(* Check Setup Level with active key switch and an active movement *)
	IF xReset THEN
		xReset:=FALSE;
		xActivateOverlayMessage:=FALSE;
	END_IF;
	IF NOT(xActivateOverlayMessage) THEN
		xActiveSetupLevel:=	(T_Visu.ptrT_ExchgParam^.T_Visu.bActivSpecialLayer <> 0) AND
							T_StartUp.T_State.xCompleted AND NOT(T_StartUp.T_State.xBlockChangeMovementVisu);
		xDoNotCheckMovement:=	NOT(T_Process.xEnd) AND NOT(T_Process.xError) AND ((T_Process.iFunctNr = 10) OR (T_Process.iFunctNr = 20) OR (T_Process.iFunctNr = 30));
		xActiveProcess:=		NOT(T_Process.xEnd) AND NOT(T_Process.xError) AND (T_Process.iFunctNr = 40);
		xActiveStation:=		NOT(T_Station.TControl.xEnd) AND NOT(T_Station.TControl.xError) AND NOT(xActiveProcess) AND NOT(xDoNotCheckMovement);
		xActiveHWStation:=	T_Station.TControl.xActiveMovement AND NOT(xActiveProcess) AND NOT(xActiveStation) AND NOT(xDoNotCheckMovement);
		(* check if the ToolTorque was activatet *)
		xStopAxisWithStationFunction:=FALSE;
		IF xActiveHWStation THEN
			IF (T_Visu.T_PlcParam.dwActualPage = 220) THEN
				xActiveHWStation:=FALSE;
				xStopAxisWithStationFunction:=TRUE;
			END_IF;
		END_IF;
	END_IF;
	FallingEdgeKeySwitchOff(CLK:=xKeySwitch);
	IF xActiveSetupLevel THEN
		IF FallingEdgeKeySwitchOff.Q THEN
			IF xActiveProcess OR xActiveStation OR xActiveHWStation OR xStopAxisWithStationFunction THEN
				xActivateOverlayMessage:=TRUE;
				iStepSwitchMachineLevel:=1;
			END_IF;
		END_IF;
	END_IF;
(*
	IF NOT(xBlockChecking) THEN
		xActivateOverlayMessage:= xActivateOverlayMessage AND NOT
								(T_Station.TControl.xSecurityCircuitOff OR T_Station.TControl.xSecurityCircuitOn);
	END_IF;
*)
	IF xActivateOverlayMessage THEN
		CASE iStepSwitchMachineLevel OF
		1:	TONWaitTimeStateMachine(IN:=FALSE);
			(* next step *)
			iStepSwitchMachineLevel:=10;
		10:	TONWaitTimeStateMachine(IN:=TRUE,PT:=T#150ms);
			IF TONWaitTimeStateMachine.Q THEN
				TONWaitTimeStateMachine(IN:=FALSE);
				(* next step *)
				iStepSwitchMachineLevel:=20;
			END_IF;
		20:	IF T_TwinSafeOut.QxContactor_K3 AND T_TwinSafeOut.QxContactor_K4 THEN
				xPowerSupplyActive:=TRUE;
				T_Visu.ptrT_ExchgParam^.T_Visu.T_Message.iState:=121;	(* Display message -> The Movement of the machine will be breaked! *)
				(* with switching off of the key switch the power supply is not switched off and the movement are still active *)
				IF xActiveProcess THEN
					T_Process.xStop:=TRUE;
					iStepSwitchMachineLevel:=30;
				END_IF;
				IF xActiveStation THEN
					T_Station.TControl.xStop:=TRUE;
					iStepSwitchMachineLevel:=40;
				END_IF;
				IF xActiveHWStation THEN
					iStepSwitchMachineLevel:=60;
				END_IF;
				IF xStopAxisWithStationFunction THEN
					iStepSwitchMachineLevel:=70;
				END_IF;
			ELSE
				(* with switching off of the key switch the power supply is switched off *)
				xPowerSupplyActive:=FALSE;
				(* next step *)
				iStepSwitchMachineLevel:=80;
			END_IF;
		30:	IF T_Process.xEnd THEN
				(* next step *)
				iStepSwitchMachineLevel:=80;
			END_IF;
			IF NOT(T_TwinSafeOut.QxContactor_K3) OR NOT(T_TwinSafeOut.QxContactor_K4) THEN
				xPowerSupplyActive:=FALSE;
				iStepSwitchMachineLevel:=80;
			END_IF;
			T_Visu.ptrT_ExchgParam^.T_Visu.T_Message.iState:=121;	(* Display message -> The Movement of the machine will be breaked! *)
		40:	IF T_Station.TControl.xEnd THEN
				(* next step *)
				T_Station.TControl.xStop:=FALSE;
				iStepSwitchMachineLevel:=60;
			END_IF;
			IF NOT(T_TwinSafeOut.QxContactor_K3) OR NOT(T_TwinSafeOut.QxContactor_K4) THEN
				xPowerSupplyActive:=FALSE;
				iStepSwitchMachineLevel:=80;
			END_IF;
			T_Visu.ptrT_ExchgParam^.T_Visu.T_Message.iState:=121;	(* Display message -> The Movement of the machine will be breaked! *)
		60:	IF T_Station.THardware.TAxisToolLeft.T_CtrleSingle.xDone AND NOT(T_Station.THardware.TAxisToolLeft.T_CtrleSingle.xErr) THEN
				T_Station.THardware.TAxisToolLeft.T_CtrleSingle.iFunction:=5;
				T_Station.THardware.TAxisToolLeft.T_CtrleSingle.xExecute:=TRUE;
			END_IF;
			IF NOT(T_Station.THardware.TAxisToolLeft.T_CtrleSingle.xDone) AND T_Station.THardware.TAxisToolLeft.T_CtrleSingle.xNotMoving AND NOT(T_Station.THardware.TAxisToolLeft.T_CtrleSingle.xErr) THEN
				T_Station.THardware.TAxisToolLeft.T_CtrleSingle.xReset:=TRUE;
			END_IF;
			IF T_Station.THardware.TAxisToolRight.T_CtrleSingle.xDone AND NOT(T_Station.THardware.TAxisToolRight.T_CtrleSingle.xErr) THEN
				T_Station.THardware.TAxisToolRight.T_CtrleSingle.iFunction:=5;
				T_Station.THardware.TAxisToolRight.T_CtrleSingle.xExecute:=TRUE;
			END_IF;
			IF NOT(T_Station.THardware.TAxisToolRight.T_CtrleSingle.xDone) AND T_Station.THardware.TAxisToolRight.T_CtrleSingle.xNotMoving AND NOT(T_Station.THardware.TAxisToolRight.T_CtrleSingle.xErr) THEN
				T_Station.THardware.TAxisToolRight.T_CtrleSingle.xReset:=TRUE;
			END_IF;
			IF T_Station.THardware.TAxisToolCenter.T_CtrleSingle.xDone AND NOT(T_Station.THardware.TAxisToolCenter.T_CtrleSingle.xErr) THEN
				T_Station.THardware.TAxisToolCenter.T_CtrleSingle.iFunction:=5;
				T_Station.THardware.TAxisToolCenter.T_CtrleSingle.xExecute:=TRUE;
			END_IF;
			IF NOT(T_Station.THardware.TAxisToolCenter.T_CtrleSingle.xDone) AND T_Station.THardware.TAxisToolCenter.T_CtrleSingle.xNotMoving AND NOT(T_Station.THardware.TAxisToolCenter.T_CtrleSingle.xErr) THEN
				T_Station.THardware.TAxisToolCenter.T_CtrleSingle.xReset:=TRUE;
			END_IF;
			IF T_Station.THardware.TAxisToolFeeder.T_CtrleSingle.xDone AND NOT(T_Station.THardware.TAxisToolFeeder.T_CtrleSingle.xErr) THEN
				T_Station.THardware.TAxisToolFeeder.T_CtrleSingle.iFunction:=5;
				T_Station.THardware.TAxisToolFeeder.T_CtrleSingle.xExecute:=TRUE;
			END_IF;
			IF NOT(T_Station.THardware.TAxisToolFeeder.T_CtrleSingle.xDone) AND NOT(T_Station.THardware.TAxisToolFeeder.T_CtrleSingle.xNotMoving) AND NOT(T_Station.THardware.TAxisToolFeeder.T_CtrleSingle.xErr) THEN
				T_Station.THardware.TAxisToolFeeder.T_CtrleSingle.iFunction:=5;
				T_Station.THardware.TAxisToolFeeder.T_CtrleSingle.xExecute:=TRUE;
			END_IF;
			IF NOT(T_Station.THardware.TAxisToolFeeder.T_CtrleSingle.xDone) AND T_Station.THardware.TAxisToolFeeder.T_CtrleSingle.xNotMoving AND NOT(T_Station.THardware.TAxisToolFeeder.T_CtrleSingle.xErr) THEN
				T_Station.THardware.TAxisToolFeeder.T_CtrleSingle.xReset:=TRUE;
			END_IF;
			IF T_Station.THardware.TAxisGrindFeeder.T_CtrleSingle.xDone AND NOT(T_Station.THardware.TAxisGrindFeeder.T_CtrleSingle.xErr) THEN
				T_Station.THardware.TAxisGrindFeeder.T_CtrleSingle.iFunction:=5;
				T_Station.THardware.TAxisGrindFeeder.T_CtrleSingle.xExecute:=TRUE;
			END_IF;
			IF NOT(T_Station.THardware.TAxisGrindFeeder.T_CtrleSingle.xDone) AND NOT(T_Station.THardware.TAxisGrindFeeder.T_CtrleSingle.xNotMoving) AND NOT(T_Station.THardware.TAxisGrindFeeder.T_CtrleSingle.xErr) THEN
				T_Station.THardware.TAxisGrindFeeder.T_CtrleSingle.iFunction:=5;
				T_Station.THardware.TAxisGrindFeeder.T_CtrleSingle.xExecute:=TRUE;
			END_IF;
			IF NOT(T_Station.THardware.TAxisGrindFeeder.T_CtrleSingle.xDone) AND T_Station.THardware.TAxisGrindFeeder.T_CtrleSingle.xNotMoving AND NOT(T_Station.THardware.TAxisGrindFeeder.T_CtrleSingle.xErr) THEN
				T_Station.THardware.TAxisGrindFeeder.T_CtrleSingle.xReset:=TRUE;
			END_IF;
			IF NOT(T_Station.THardware.TCylToolTension.T_CtrleCyl.xDone) THEN T_Station.THardware.TCylToolTension.T_CtrleCyl.xReset:=TRUE; END_IF;
			T_Visu.ptrT_ExchgParam^.T_Visu.T_Message.iState:=121;	(* Display message -> The Movement of the machine will be breaked! *)
			(* next step *)
			iStepSwitchMachineLevel:=80;
		70:	IF T_Station.TControl.xEnd THEN
				(* next step *)
				T_Station.TControl.iFunctNr:=3;
				T_Station.TControl.xStart:=TRUE;
				iStepSwitchMachineLevel:=71;
			END_IF;
			IF NOT(T_TwinSafeOut.QxContactor_K3) OR NOT(T_TwinSafeOut.QxContactor_K4) THEN
				xPowerSupplyActive:=FALSE;
				iStepSwitchMachineLevel:=80;
			END_IF;
			T_Visu.ptrT_ExchgParam^.T_Visu.T_Message.iState:=121;	(* Display message -> The Movement of the machine will be breaked! *)
		71:	IF NOT(T_Station.TControl.xStart) AND T_Station.TControl.xEnd THEN
				(* next step *)
				iStepSwitchMachineLevel:=80;
			END_IF;
			IF NOT(T_TwinSafeOut.QxContactor_K3) OR NOT(T_TwinSafeOut.QxContactor_K4) THEN
				xPowerSupplyActive:=FALSE;
				iStepSwitchMachineLevel:=80;
			END_IF;
		80:	IF NOT(T_Visu.T_CtrleVisu.xExecute) AND T_Visu.T_CtrleVisu.xDone THEN
				T_Visu.ptrT_ExchgParam^.T_Visu.T_Message.iState:=0;
				T_Visu.ptrT_ExchgParam^.T_Visu.bActivSpecialLayer:=0;
				T_Visu.ptrT_ExchgParam^.T_TouchScreenBtPanel.iStateBtLeft:=0;
				T_Visu.ptrT_ExchgParam^.T_TouchScreenNavPanel.wState:=1;
				T_Visu.T_PlcParam.dwSetNewPage:=16#A;	(* Main Page wird aufgerufen *)
				T_Visu.T_CtrleVisu.iFunction:=1;
				T_Visu.T_CtrleVisu.xExecute:=TRUE;
				iStepSwitchMachineLevel:=90;
			END_IF;
		90:	IF NOT(T_Visu.T_CtrleVisu.xExecute) AND T_Visu.T_CtrleVisu.xDone THEN
				T_StartUp.T_State.xBlockChangeMovementVisu:=TRUE;	(* Lock the navigation of the visu *)
				T_Visu.ptrT_ExchgParam^.T_SafetyCtrl.xBlockVisuObject:=TRUE;
				T_StartUp.T_State.xBlockVisuNavigation:=FALSE;	(* Unlock the navigation of the visu *)
				T_Visu.ptrT_ExchgParam^.T_SafetyCtrl.bStateAutoGeometry:=1;
				T_Visu.ptrT_ExchgParam^.T_SafetyCtrl.bStateAutoGroove:=1;
				T_Visu.ptrT_ExchgParam^.T_SafetyCtrl.bStateReference:=1;
				T_Visu.ptrT_ExchgParam^.T_SafetyCtrl.bStateToolCalibration:=1;
				T_Visu.ptrT_ExchgParam^.T_SafetyCtrl.bStateToolTorque:=1;
				T_Visu.ptrT_ExchgParam^.T_SafetyCtrl.bStateTeachInToolLeft:=1;
				T_Visu.ptrT_ExchgParam^.T_SafetyCtrl.bStateTeachInToolCenter:=1;
				T_Visu.ptrT_ExchgParam^.T_SafetyCtrl.bStateTeachInToolRight:=1;
				T_Visu.ptrT_ExchgParam^.T_SafetyCtrl.bStateTeachInToolFeeder:=1;
				T_Visu.ptrT_ExchgParam^.T_SafetyCtrl.bStateTeachInGrindFeeder:=1;
				T_Visu.ptrT_ExchgParam^.T_StationCommon.iWireFeederRefIndexState:=1;
				(* Overlay Message Error *)
				T_Visu.ptrT_ExchgParam^.T_SafetyCtrl.bStateMessageError:=1;
				T_Visu.ptrT_ExchgParam^.T_SafetyCtrl.bStateMessageInfo:=0;
				T_Visu.ptrT_ExchgParam^.T_SafetyCtrl.bStateMessageWarning:=0;
				IF xPowerSupplyActive THEN
					T_Visu.ptrT_ExchgParam^.T_SafetyCtrl.iMsgErrorLine1:=18;	(* WHILE A MOVEMENT THE KEY SWITCH *)
					T_Visu.ptrT_ExchgParam^.T_SafetyCtrl.iMsgErrorLine2:=18;	(* HAS BEEN SWITCHED OFF! *)
					T_Visu.ptrT_ExchgParam^.T_SafetyCtrl.iMsgErrorLine3:=18;	(* NOW YOU ARE ON THE NORMAL OPERATION *)
					T_Visu.ptrT_ExchgParam^.T_SafetyCtrl.iMsgErrorLine4:=18;	(* AND THE POWER SUPPLY IS STILL SWITCHED ON *)
					T_Visu.ptrT_ExchgParam^.T_SafetyCtrl.xConfirmMsgError:=FALSE;
				ELSE
					T_Visu.ptrT_ExchgParam^.T_SafetyCtrl.iMsgErrorLine1:=17;	(* WHILE A MOVEMENT THE KEY SWITCH *)
					T_Visu.ptrT_ExchgParam^.T_SafetyCtrl.iMsgErrorLine2:=17;	(* HAS BEEN SWITCHED OFF! *)
					T_Visu.ptrT_ExchgParam^.T_SafetyCtrl.iMsgErrorLine3:=17;	(* NOW YOU ARE ON THE NORMAL OPERATION *)
					T_Visu.ptrT_ExchgParam^.T_SafetyCtrl.iMsgErrorLine4:=17;	(* AND THE POWER SUPPLY IS SWITCHED OFF *)
					T_Visu.ptrT_ExchgParam^.T_SafetyCtrl.xConfirmMsgError:=FALSE;
				END_IF;
				(* next step *)
				iStepSwitchMachineLevel:=100;
			END_IF;
		100:	IF T_Visu.ptrT_ExchgParam^.T_SafetyCtrl.xConfirmMsgError THEN
				T_StartUp.T_State.xBlockChangeMovementVisu:=FALSE;	(* Unlock the navigation of the visu *)
				T_Visu.ptrT_ExchgParam^.T_SafetyCtrl.xBlockVisuObject:=FALSE;
				T_StartUp.T_State.xBlockVisuNavigation:=FALSE;	(* Unlock the navigation of the visu *)
				T_Visu.ptrT_ExchgParam^.T_SafetyCtrl.bStateAutoGeometry:=1;
				T_Visu.ptrT_ExchgParam^.T_SafetyCtrl.bStateAutoGroove:=1;
				T_Visu.ptrT_ExchgParam^.T_SafetyCtrl.bStateReference:=1;
				T_Visu.ptrT_ExchgParam^.T_SafetyCtrl.bStateToolCalibration:=1;
				T_Visu.ptrT_ExchgParam^.T_SafetyCtrl.bStateToolTorque:=1;
				T_Visu.ptrT_ExchgParam^.T_SafetyCtrl.bStateTeachInToolLeft:=1;
				T_Visu.ptrT_ExchgParam^.T_SafetyCtrl.bStateTeachInToolCenter:=1;
				T_Visu.ptrT_ExchgParam^.T_SafetyCtrl.bStateTeachInToolRight:=1;
				T_Visu.ptrT_ExchgParam^.T_SafetyCtrl.bStateTeachInToolFeeder:=1;
				T_Visu.ptrT_ExchgParam^.T_SafetyCtrl.bStateTeachInGrindFeeder:=1;
				T_Visu.ptrT_ExchgParam^.T_StationCommon.iWireFeederRefIndexState:=1;
				T_Visu.ptrT_ExchgParam^.T_SafetyCtrl.bStateMessageError:=0;
				T_Visu.ptrT_ExchgParam^.T_SafetyCtrl.xConfirmMsgError:=FALSE;
				xActivateOverlayMessage:=FALSE;
				iStepSwitchMachineLevel:=1;
			END_IF;
			IF NOT(T_TwinSafeOut.QxContactor_K3) OR NOT(T_TwinSafeOut.QxContactor_K4) THEN
				T_Visu.ptrT_ExchgParam^.T_SafetyCtrl.iMsgErrorLine1:=17;	(* WHILE A MOVEMENT THE KEY SWITCH *)
				T_Visu.ptrT_ExchgParam^.T_SafetyCtrl.iMsgErrorLine2:=17;	(* HAS BEEN SWITCHED OFF! *)
				T_Visu.ptrT_ExchgParam^.T_SafetyCtrl.iMsgErrorLine3:=17;	(* NOW YOU ARE ON THE NORMAL OPERATION *)
				T_Visu.ptrT_ExchgParam^.T_SafetyCtrl.iMsgErrorLine4:=17;	(* AND THE POWER SUPPLY IS SWITCHED OFF *)
			END_IF;
			IF T_TwinSafeOut.QxContactor_K3 AND T_TwinSafeOut.QxContactor_K4  THEN
				T_Visu.ptrT_ExchgParam^.T_SafetyCtrl.iMsgErrorLine1:=18;	(* WHILE A MOVEMENT THE KEY SWITCH *)
				T_Visu.ptrT_ExchgParam^.T_SafetyCtrl.iMsgErrorLine2:=18;	(* HAS BEEN SWITCHED OFF! *)
				T_Visu.ptrT_ExchgParam^.T_SafetyCtrl.iMsgErrorLine3:=18;	(* NOW YOU ARE ON THE NORMAL OPERATION *)
				T_Visu.ptrT_ExchgParam^.T_SafetyCtrl.iMsgErrorLine4:=18;	(* AND THE POWER SUPPLY IS STILL SWITCHED ON *)
			END_IF;
		END_CASE;
	END_IF;
END_FUNCTION_BLOCK

(* POU PRG_VISU_LAYER5/PRG_VISU, FBD *)
PROGRAM PRG_VISU
VAR
	fbVisuQVis: FBQVIS;
	xSecurityKey: BOOL;
	FBCtrleButton: FB_CTRLEBUTTON;
END_VAR
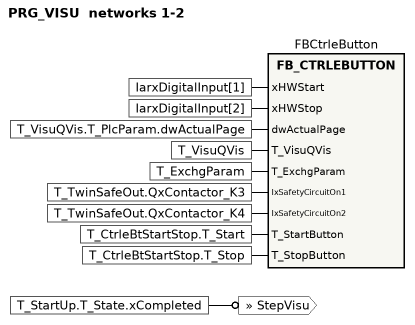
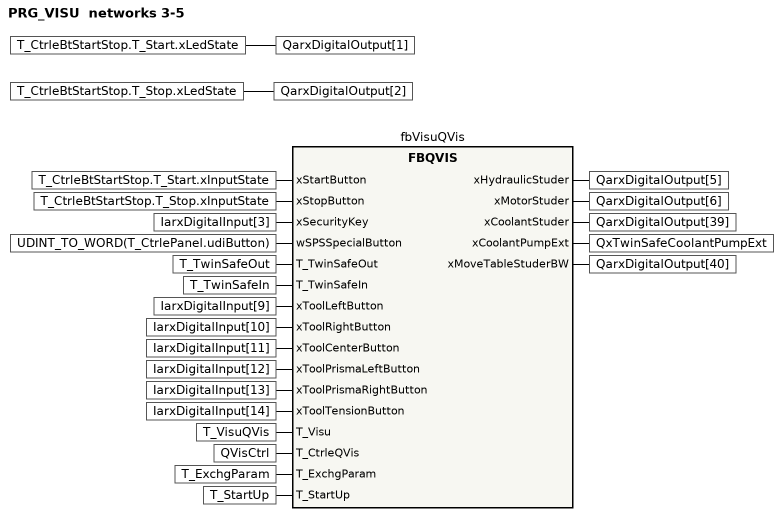
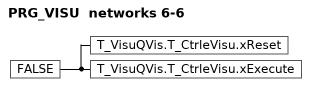
_FBD_ (* Function Block Diagram *)
NETWORK 1 (* VISUALISATION LEVEL-->LAYER 5 *)
	FBCtrleButton:FB_CTRLEBUTTON(xHWStart: IarxDigitalInput[1], xHWStop: IarxDigitalInput[2], dwActualPage: T_VisuQVis.T_PlcParam.dwActualPage, T_VisuQVis: T_VisuQVis, T_ExchgParam: T_ExchgParam, IxSafetyCircuitOn1: T_TwinSafeOut.QxContactor_K3, IxSafetyCircuitOn2: T_TwinSafeOut.QxContactor_K4, T_StartButton: T_CtrleBtStartStop.T_Start, T_StopButton: T_CtrleBtStartStop.T_Stop)
NETWORK 2
	NOT T_StartUp.T_State.xCompleted => >>StepVisu
NETWORK 3
	T_CtrleBtStartStop.T_Start.xLedState => QarxDigitalOutput[1]
NETWORK 4
	T_CtrleBtStartStop.T_Stop.xLedState => QarxDigitalOutput[2]
NETWORK 5 StepVisu:
	fbVisuQVis:FBQVIS(xStartButton: T_CtrleBtStartStop.T_Start.xInputState, xStopButton: T_CtrleBtStartStop.T_Stop.xInputState, xSecurityKey: IarxDigitalInput[3], wSPSSpecialButton: UDINT_TO_WORD(T_CtrlePanel.udiButton), T_TwinSafeOut: T_TwinSafeOut, T_TwinSafeIn: T_TwinSafeIn, xToolLeftButton: IarxDigitalInput[9], xToolRightButton: IarxDigitalInput[10], xToolCenterButton: IarxDigitalInput[11], xToolPrismaLeftButton: IarxDigitalInput[12], xToolPrismaRightButton: IarxDigitalInput[13], xToolTensionButton: IarxDigitalInput[14], T_Visu: T_VisuQVis, T_CtrleQVis: QVisCtrl, T_ExchgParam: T_ExchgParam, T_StartUp: T_StartUp, xMotorStuder => QarxDigitalOutput[6], xCoolantStuder => QarxDigitalOutput[39], xCoolantPumpExt => QxTwinSafeCoolantPumpExt, xMoveTableStuderBW => QarxDigitalOutput[40]) => QarxDigitalOutput[5]
NETWORK 6
	FALSE => T_VisuQVis.T_CtrleVisu.xReset, T_VisuQVis.T_CtrleVisu.xExecute
_END_FBD_
(* the same logic as Structured Text *)
(* Network 1: VISUALISATION LEVEL-->LAYER 5 *)
FBCtrleButton(xHWStart := IarxDigitalInput[1], xHWStop := IarxDigitalInput[2], dwActualPage := T_VisuQVis.T_PlcParam.dwActualPage, T_VisuQVis := T_VisuQVis, T_ExchgParam := T_ExchgParam, IxSafetyCircuitOn1 := T_TwinSafeOut.QxContactor_K3, IxSafetyCircuitOn2 := T_TwinSafeOut.QxContactor_K4, T_StartButton := T_CtrleBtStartStop.T_Start, T_StopButton := T_CtrleBtStartStop.T_Stop);
(* Network 2 *)
IF NOT T_StartUp.T_State.xCompleted THEN JMP StepVisu; END_IF;
(* Network 3 *)
QarxDigitalOutput[1] := T_CtrleBtStartStop.T_Start.xLedState;
(* Network 4 *)
QarxDigitalOutput[2] := T_CtrleBtStartStop.T_Stop.xLedState;
(* Network 5 *)
StepVisu:
fbVisuQVis(xStartButton := T_CtrleBtStartStop.T_Start.xInputState, xStopButton := T_CtrleBtStartStop.T_Stop.xInputState, xSecurityKey := IarxDigitalInput[3], wSPSSpecialButton := UDINT_TO_WORD(T_CtrlePanel.udiButton), T_TwinSafeOut := T_TwinSafeOut, T_TwinSafeIn := T_TwinSafeIn, xToolLeftButton := IarxDigitalInput[9], xToolRightButton := IarxDigitalInput[10], xToolCenterButton := IarxDigitalInput[11], xToolPrismaLeftButton := IarxDigitalInput[12], xToolPrismaRightButton := IarxDigitalInput[13], xToolTensionButton := IarxDigitalInput[14], T_Visu := T_VisuQVis, T_CtrleQVis := QVisCtrl, T_ExchgParam := T_ExchgParam, T_StartUp := T_StartUp);
QarxDigitalOutput[6] := fbVisuQVis.xMotorStuder;
QarxDigitalOutput[39] := fbVisuQVis.xCoolantStuder;
QxTwinSafeCoolantPumpExt := fbVisuQVis.xCoolantPumpExt;
QarxDigitalOutput[40] := fbVisuQVis.xMoveTableStuderBW;
QarxDigitalOutput[5] := fbVisuQVis.xHydraulicStuder;
(* Network 6 *)
T_VisuQVis.T_CtrleVisu.xReset := FALSE;
T_VisuQVis.T_CtrleVisu.xExecute := FALSE;
END_PROGRAM

(* POU PRG_VISU_LAYER5/FB_VISU/FBQVIS, ST *)
FUNCTION_BLOCK FBQVIS
VAR_INPUT
	xStartButton:BOOL;					(* external start button *)
	xStopButton:BOOL;					(* external stop button *)
	xSecurityKey:BOOL;					(* state of the keyswitch *)
	wSPSSpecialButton:WORD;			(* input of the special button of the controlpanel *)
	T_TwinSafeOut:ST_TWINSAFE_OUT;	(* Output of the TwinSAFE components *)
	T_TwinSafeIn:ST_TWINSAFE_IN;		(* Input of the TwinSAFE components *)
(*22.12.2009: KFS	{	*)
	xToolLeftButton:BOOL;					(* Signal of the button for closing the ToolLeft-->this is only for the MicroRod *)
	xToolRightButton:BOOL;				(* Signal of the button for closing the ToolRight-->this is only for the MicroRod *)
	xToolCenterButton:BOOL;				(* Signal of the button for closing the ToolCenter-->this is only for the MicroRod *)
	xToolPrismaLeftButton:BOOL;			(* Signal of the button for closing the ToolPrismaLeft-->this is only for the MicroRod *)
	xToolPrismaRightButton:BOOL;			(* Signal of the button for closing the ToolPrismaRight-->this is only for the MicroRod *)
	xToolTensionButton:BOOL;				(* Signal of the button for activate the ToolTension-->this is only for the MicroRod *)
(*22.12.2009: KFS	}	*)
END_VAR
VAR_OUTPUT
(* SOA 02.02.2023     {     *)
	xHydraulicStuder: 	BOOL;  					(*Hydraulic Pump of Studer S20 Machine*)
	xMotorStuder: BOOL;						(*Grinding-Engine of Studer S20 Machine*)
	xCoolantStuder: BOOL;						(*Coolant Pump of Studer S20 Machine*)
	xCoolantPumpExt: BOOL;					(*Coolant Pump external*)
	xMoveTableStuderBW:BOOL;
(* SOA 02.02.2023    }   *)
END_VAR
VAR_IN_OUT
	T_Visu:ST_QVIS;
	T_CtrleQVis:ST_QVISCTRLE;
	T_ExchgParam:ST_QVIS_EXCHG_PARAM;
	T_StartUp:ST_STARTUP;
END_VAR
VAR
	RisingEdgeActiv:R_TRIG;
	RisingEdgeExecute:R_TRIG;
	RisingEdgeExecuteAction:R_TRIG;
	RisingEdgeBtPanelLeft:R_TRIG;
	FallingEdgeBtPanelLeft:F_TRIG;
	RisingEdgeSpecialLayer:R_TRIG;
	FallingEdgeSpecialLayer:F_TRIG;
	RisingEdgeTouchScreenNavPanel:R_TRIG;
	FallingEdgeTouchScreenNavPanel:F_TRIG;
	RisingEdgeBtPanelRight:R_TRIG;
	FallingEdgeBtPanelRight:F_TRIG;
	RisingEdgeBtFunctionPanel:R_TRIG;
	FallingEdgeBtFunctionPanel:F_TRIG;
	RisingEdgeDynPassword:R_TRIG;
	RisingEdgeGeometryManagement:R_TRIG;
	RisingEdgeToolDiameter:R_TRIG;
	RisingEdgePrisma:R_TRIG;
	xChangePage:BOOL:=FALSE;
	dwInCount_QVisCmd:DWORD:=0;
	xTmp: BOOL;
	wActivBtLeft: WORD;
	wActivBtRight: WORD;
	fbQvisInitPage:FBQVIS_INITPAGE;
	xNavPanelChangePage: BOOL;
	xBtPanelLeftChangePage:BOOL;
	xBtPanelRightChangePage: BOOL; (*SOA*)
	xNextPageVertical:BOOL;
	xSetParameterPage:BOOL;
	xActivationSection1: BOOL;
	xActivationSection2: BOOL;
	xActivationSection3: BOOL;
	xActivationSection4: BOOL;
	xActivationSection5: BOOL; (*SOA *)
	xActivationSection6: BOOL; (*SOA *)

	xSetPitchEqual: BOOL;
	iStepAction: INT;
	xStepActionDone: BOOL;
	bOldActivSpecialLayer: BYTE;
	wSpecialLayerGeneralActivTask: WORD;
	wSpecialLayerToolRotActivTask: WORD;
	wSpecialLayerWireFeedActivTask: WORD;
	wSpecialLayerGrindAxisActivTask: WORD;
	wSpecialLayerGeneralActivPage: WORD;
	wSpecialLayerToolRotActivPage: WORD;
	wSpecialLayerWireFeedActivPage: WORD;
	wSpecialLayerGrindAxisActivPage: WORD;
	dwSetNewPage: DWORD;
	wNormalLayerActivTask: WORD;
	wNormalLayerActivPage: WORD;
	ii: INT;
	wTmp: WORD;
	awNormalLayerActivPage:ARRAY [1..6] OF WORD;
	awSpecialLayerGeneralActivPage:ARRAY [1..6] OF WORD;
	awSpecialLayerToolRotActivPage:ARRAY [1..6] OF WORD;
	awSpecialLayerWireFeedActivPage:ARRAY [1..6] OF WORD;
	awSpecialLayerGrindAxisActivPage:ARRAY [1..6] OF WORD;
	wTmpNormalLayerActivTask: WORD;
	wTmpSpecialLayerGeneralActivTask: WORD;
	wTmpSpecialLayerToolRotActivTask: WORD;
	wTmpSpecialLayerWireFeedActivTask: WORD;
	wTmpSpecialLayerGrindAxisActivTask: WORD;
	wStandardPageNr: WORD;
	iTmpActivBtLeft: INT;
	(* Random *)
	fbGetCpuAccount:GETCPUCOUNTER;
	fbPwSystem:FBPW_SYSTEM;
	(* Pw *)
	iPwSystem:INT;
	iStepCounter: INT;
	arSaveToolGeometry:ST_GEOMETRY;
	rSectionPitch: REAL;
	ptxActiveSection1: POINTER TO BOOL;
	ptxActiveSection2: POINTER TO BOOL;
	ptxActiveSection3: POINTER TO BOOL;
	ptxActiveSection4: POINTER TO BOOL;
	ptxActiveSection5: POINTER TO BOOL;
	ptxActiveSection6: POINTER TO BOOL;

	xOverlayMeasureToolDia: BOOL;
	xPlungeActivation: BOOL;
	xDisplaceActivation: BOOL;
	xCorrectionToolDiameterAdd: BOOL;
	xCorrectionToolDiameterAddMore: BOOL;
	xCorrectionToolDiameterSub: BOOL;
	xCorrectionToolDiameterSubMore: BOOL;
	xResetToolDiameterCorrection: BOOL;
	xKeyPadActivation: BOOL;
	xFctCorrectionToolDiameter: BOOL;
	rCorrectionValue: REAL;

(* Key panel button "Esc"/"Enter" *)
	RisingEdgeKeyPanel_Esc:R_TRIG;
	RisingEdgeKeyPanel_Enter:R_TRIG;
(*22.12.2009: KFS	{	 *)
(* External button for the tool-clamping*)
	RisingEdgeBtToolLeft:R_TRIG;
	RisingEdgeBtToolRight:R_TRIG;
	RisingEdgeBtToolCenter:R_TRIG;
	RisingEdgeBtToolPrismaLeft:R_TRIG;
	RisingEdgeBtToolPrismaRight:R_TRIG;
	RisingEdgeBtToolTension:R_TRIG;
(*22.12.2009: KFS	}	 *)
(* variable start action *)
	TimerAction:TON;
	TimerNotReady:TOF;
	tTimeOutAction:TIME;
	xSelectPrisma: BOOL;
	xToolTensForceAdd: BOOL;
	xToolTensForceAddMore: BOOL;
	xToolTensForceSub: BOOL;
	xToolTensForceSubMore: BOOL;
	xResetCalculToolRotTorque: BOOL;
	rCalcTotalToolLength: REAL;
	xTmpSecurityKey: BOOL;
	RisingEdgeTemp:R_TRIG;
	TONWAIT: TON;
	xPart1: BOOL;
	xPart2: BOOL;
	xPart3: BOOL;
	xPart4: BOOL;
	xPart5: BOOL;
	xPart6: BOOL;

	iPartActive: INT;
	xToolRotationMasterSlave: BOOL;
	xSwitchMasterSlave: BOOL;
	xQvisActiv: BOOL;
	TimerQVis: TON;
	RisingEdgeReset:R_TRIG;
	xConfirmResetFB: BOOL;
	xFirstRead: BOOL;
	ptrTeachINAxis:POINTER TO ST_AXIS;
	ptrCylAction:POINTER TO ST_CYLINDER;
	xStopAxis: BOOL;
	xMoveRelPosition: BOOL;
	TParaAxisTeachIN:ST_EXCHG_PARAM_TEACHIN;
	xMoveContinousVel: BOOL;
	xMoveAbsPosition: BOOL;
	bButtonPanelLocked: BYTE;
	xDelayActionBtPanelRight: BOOL;
	TimerPressBtPanelRight: TON;

(* Structure page *)
	T_ConfigPage:ST_CONFIGPAGE;
	wMaskBtPanelLeft: WORD;
	wMaskBtPanelRight: WORD;
	wMaskFunctionPanel: WORD;
	RisingEdgeProcessDone: R_TRIG;
	xStopImmediatly: BOOL;
	RisingEdgeProcessError: R_TRIG;
	RisingEdgeResetProcess: R_TRIG;
	RisingEdgeExecuteProcess: R_TRIG;
	RisingEdgeActionNotReady: R_TRIG;
	FallingEdgeActionNotReady: F_TRIG;
	RisingEdgeActionDone: R_TRIG;
	xBlockConfirmMessage: BOOL;
	RisingEdgeActionError: R_TRIG;
	RisingEdgeResetAction: R_TRIG;
	xSlowFast: BOOL;
	iSelectedAxis: INT;
	xSlowFastJogToolRotation: BOOL;
	xSlowFastJogToolFeeder: BOOL;
	xSlowFastJogGrindFeeder: BOOL;
	xToggleAxisPower: BOOL;
	xResetAxis: BOOL;
	xUpdateProfileList: BOOL;
	jj: INT;
	RisingEdgePtrProfileListUpDown: R_TRIG;
	iPointerListProfile: INT;
	iActualActiveProfile: INT;
	xAction_CopyProfileToProcess: BOOL;
	xProfileFileNotFound: BOOL;
	iToLoadProfileNr: INT;
	sToLoadProfileName: STRING;
	sTmpDynamicText: STRING;
	xAction_LoadProfileToProcessImage: BOOL;
	xAction_SaveNovRAM: BOOL;
	xActionDeleteProfile: BOOL;
	TimerONTmp: TON;
	iStepActionNovRam: INT;
	xAction_SaveProfileToFile: BOOL;
	iTmp: INT;
	sTmp: STRING;
	sTmp_2: STRING;
	RisingEdgeTimeOut: R_TRIG;
	fbCompareProfileProcessValue:FB_COMPAREPROFILEPROCESSVALUE;
	FailingEdgeGeometryManagement: F_TRIG;
	FailingEdgePrisma: F_TRIG;
	rCalcMinMaxToolDia: REAL;
	xResetParaListValue: BOOL;
	xActivateStationFunction: BOOL;
	iTmpStationFunctionNr: INT;
	xFirstReadInit: BOOL;
	xFirstReadReset: BOOL;
	xMicroRodActive: BOOL;
	FBCalcTorqueToolLeft: FB_CALC_TORQUE;
	FBCalcTorqueToolCenter: FB_CALC_TORQUE;
	FBCalcTorqueToolRight: FB_CALC_TORQUE;
	xTmpStopAxis: BOOL;
	RisingEdgeStartButton: R_TRIG;
	dwPageNrProcessStart: DWORD;
	FallingEdgeStartButton: F_TRIG;
	RisingEdgeStopButton: R_TRIG;
	FallingEdgeStopButton: F_TRIG;
	xToggleCylinderState: BOOL;
	dwTmpActualPage: DWORD;
	xUpdateErrorList: BOOL;
	RisingEdgeErrorList: R_TRIG;
	xParameterSavedErrorList: BOOL;
	xDeleteErrorList: BOOL;
	FBQVisErrorList: FBQVIS_ERROR_LIST;
	FBSetErrorList:FB_SETERRORLIST;
	xProcessMachine: BOOL;
	xProcessStation: BOOL;
	iStepProcess: INT;
	xStepProcessDone: BOOL;
	xStopProcess: BOOL;
	xAction_StopCycle: BOOL;
	xWaitStopEnd: BOOL;
	xWaitStopCycleEnd: BOOL;
	iStepWaitStopEnd: INT;
	xActionProcStation: BOOL;
	xActionProcMachine: BOOL;
	RisingEdgeKeySwitch1: R_TRIG;
	FailingEdgeKeySwitch1: F_TRIG;
	TimerDisplayMessage: TON;
	RisingEdgeReleaseWarning: R_TRIG;
	rCalcPrismaFactor: REAL;
	xFirstReadParaList: BOOL;
	iTmpSelectParaList: INT;
	xAction_SaveNovRAMWithoutConfirm: BOOL;
	diErrorNr: DINT;
	FBErrorMessage : FB_ErrorMessage;
	fbQvisClearError:FBQVIS_CLEARERROR;
	xResetError: BOOL;
	TONTimeWaitMsg: TON;
	xCheckQuitError: BOOL;
	bStateMachine: BYTE;
	xSetStateMachine: BOOL;
	iSelectAxisToolRotation: INT;
	rAutoTimeTotal: REAL;
	rToolRotationSpeed: REAL;
	iAutoProcess: INT;
	xBlockGrindFeederActivation: BOOL;
	xToolFeederMoveStartPos: BOOL;
	xToggleAllAxisPower: BOOL;
	FBCalcProcessTime: FB_CALCPROCESSTIME;
	xReferenceAxis: BOOL;
	xTeachPosition: BOOL;
	xCalcAngleRefIndex: BOOL;
	uiToolLeftZeroTorque: UINT;
	uiToolCenterZeroTorque: UINT;
	uiToolRightZeroTorque: UINT;
	xSetCalculToolRotTorque: BOOL;
	rActualToolFeederPosition: REAL;
	xReadActualToolFeedPos: BOOL;
	xReadActualToolFeedPos1: BOOL;
	rActualToolFeederPosition1: REAL;
	rToolTotalLength: REAL;
	xCalcFirstTime: BOOL;
	xFirstReadParaList1: BOOL;
	iTmpSelectParaList1: INT;
	xTmpTeach: BOOL;
	wTmpActivBtRight: WORD;
	xOverlayGrindFeedSetPlung: BOOL;
	xOpenMessageBox: BOOL;
	lrActualGrindFeedPosition: LREAL;
	lrToWriteGrindFeedPosition: LREAL;
	xCalcAgainProcTime: BOOL;
	xToolFeederMoveLoadPos: BOOL;
	xWarmUp:BOOL;
	iSelectedCylinder: INT;
	xWarmUpMessage: BOOL;
	xWarmUpMessageActiv: BOOL;
	xWarmUpMessageDone: BOOL;

(*SOA 12.01.2023 { *)
	(*WarmUp*)
	xSaveValueWarmUp: BOOL;
	fbSetLocalTime	:NT_SetLocalTime;
	fbGetSysTime	: NT_GetTime;
	xGetTime: BOOL;
        TIMESTR :TIMESTRUCT;
	TONWaitGetTime: TON;
	xSaveTimeAndDate: BOOL;
	xInitReadFirstTimeTimeStamp: BOOL;
	iCountDayOfWeek: INT;
	xReadyToCheckWarmUp: BOOL;
	wCheckTimeWarmUp: WORD;
	wConvertMinute: WORD;
	wConertMinute_StartTime: WORD;
	wCheckTimeWarmUp_StartTime: WORD;
	wConertMinute_StopTime: WORD;
	wCheckTimeWarmUp_StopTime: WORD;
	xReadyToStartNextTime: BOOL;
	xWarmuUp_Start: BOOL;
	xWarmUp_Stop: BOOL;
	TONWarmUpChangeColour: TON;

	TONDelayMessage: TON;
	xConfirmStartWarmUp: BOOL;
	xStartUpConfirmed: BOOL;
	xStopWarmup: BOOL;
(*SOA 12.01.2023 { *)


	(* .CtrlFunctionButton *)
	wForceMaskFunctionPanel:WORD;						(* IGS *)
	aiForceRTrigActionFunctionPanel:ARRAY [1..12] OF INT;	(* IGS *)
	aiDelectRTrigActionFunctionPanel:ARRAY [1..12] OF INT;	(* IGS *)

	(* .CtrlVisuFunction *)
	xCWCCW:BOOL;										(* IGS *)
	xCylBrake:BOOL;										(* IGS *)
END_VAR
(****************************************************************************************************************************************************)
(******    This Functionblock manages the hole visualisation. It is the interface from QVis and the control application         	  *******)
(****************************************************************************************************************************************************)
	IF NOT(xFirstRead) THEN
		xFirstRead:=TRUE;
		T_Visu.ptrT_ExchgParam:=ADR(T_ExchgParam);
	END_IF;
	RisingEdgeActiv(CLK:=T_Visu.T_CtrleVisu.xActive);
	IF RisingEdgeActiv.Q THEN
		(* call functionblock init. *)
		fbQvisInitPage(T_Visu:=T_Visu);
		(* Init. variable for visualisation action *)
		T_Visu.T_CtrleAction.xDone:=TRUE;
		T_Visu.T_CtrleAction.xExecute:=FALSE;
		T_Visu.T_CtrleAction.xNotReady:=FALSE;
		T_Visu.T_CtrleAction.xErr:=FALSE;
		T_Visu.T_CtrleAction.udiErrorID:=0;
		T_Visu.T_CtrleVisu.xDone:=FALSE;
		T_Visu.ptrT_ExchgParam:=ADR(T_ExchgParam);
		wNormalLayerActivTask:=1;
		wSpecialLayerGeneralActivTask:=1;
		wSpecialLayerToolRotActivTask:=1;
		wSpecialLayerWireFeedActivTask:=1;
		wSpecialLayerGrindAxisActivTask:=1;
		wNormalLayerActivPage:=10;
		wSpecialLayerGeneralActivPage:=110;
		wSpecialLayerToolRotActivPage:=210;
		wSpecialLayerWireFeedActivPage:=310;
		wSpecialLayerGrindAxisActivPage:=410;
		T_Visu.ptrT_ExchgParam^.T_TouchScreenNavPanel.wState:=1;
		wStandardPageNr:=10;
		T_Visu.ptrT_ExchgParam^.T_Visu.T_Level.iPwSystem:=999;
		wTmpNormalLayerActivTask:=1;
		wTmpSpecialLayerGeneralActivTask:=1;
		wTmpSpecialLayerToolRotActivTask:=1;
		wTmpSpecialLayerWireFeedActivTask:=1;
		wTmpSpecialLayerGrindAxisActivTask:=1;
		FOR ii:=1 TO 6 DO
			awNormalLayerActivPage[ii]:=wStandardPageNr;
			wStandardPageNr:=wStandardPageNr + 10;
		END_FOR;
		wStandardPageNr:=110;
		FOR ii:=1 TO 6 DO
			awSpecialLayerGeneralActivPage[ii]:=wStandardPageNr;
			wStandardPageNr:=wStandardPageNr + 10;
		END_FOR;
		wStandardPageNr:=210;
		FOR ii:=1 TO 6 DO
			awSpecialLayerToolRotActivPage[ii]:=wStandardPageNr;
			wStandardPageNr:=wStandardPageNr + 10;
		END_FOR;
		wStandardPageNr:=310;
		FOR ii:=1 TO 6 DO
			awSpecialLayerWireFeedActivPage[ii]:=wStandardPageNr;
			wStandardPageNr:=wStandardPageNr + 10;
		END_FOR;
		wStandardPageNr:=410;
		FOR ii:=1 TO 6 DO
			awSpecialLayerGrindAxisActivPage[ii]:=wStandardPageNr;
			wStandardPageNr:=wStandardPageNr + 10;
		END_FOR;
		IF NOT(xFirstReadInit) THEN
			xFirstReadInit:=TRUE;
			T_Visu.T_PlcParam.dwSetNewPage:=1001;
		ELSE
			T_Visu.T_PlcParam.dwSetNewPage:=0;
		END_IF;
		T_Visu.T_PlcParam.dwActualPage:=0;
		T_Visu.T_PlcParam.dwPreviousPage:=0;
		iPointerListProfile:=1;
		iActualActiveProfile:=-1;
		TimerAction(IN:=FALSE);
		(* Init FB *)
		fbQvisClearError(	xExecute:=FALSE,
						iError:=0,
						T_Message:=T_ExchgParam.T_Visu.T_Message,
						T_Station:=T_Station,
						T_Process:=T_Process,
						T_NovRAM:=T_NovRAM,
						T_Profile:=T_Profile,
						T_HDD:=T_HDD,
						xDone=>T_Visu.T_CtrleAction.xDone,
						xNotReady=>T_Visu.T_CtrleAction.xNotReady,
						xErr=>T_Visu.T_CtrleAction.xErr,
						udiErrorID=>T_Visu.T_CtrleAction.udiErrorID);
		T_Visu.ptrT_ExchgParam^.T_Cylinder.iSelectToolTensionForce:=1;	(* For starting the machine always set  the process force for the ToolTension *)
		ptrTeachINAxis:=ADR(T_Station.THardware.TAxisToolLeft);
	END_IF;

	IF NOT (T_Visu.T_CtrleVisu.xActive) THEN
		RETURN;
	END_IF;

(* waiting for reset *)
	RisingEdgeReset(CLK:=T_Visu.T_CtrleVisu.xReset);
	IF RisingEdgeReset.Q THEN
		(* Init. structure *)
		T_Visu.T_CtrleVisu.xDone:=FALSE;
		T_Visu.T_CtrleVisu.iFunction:=0;
		T_Visu.T_CtrleVisu.xErr:=FALSE;
		T_Visu.T_CtrleVisu.udiErrorID:=0;
		IF NOT(xFirstReadReset) THEN
			xFirstReadReset:=TRUE;
			T_Visu.T_PlcParam.dwSetNewPage:=1001;
		ELSE
			T_Visu.T_PlcParam.dwSetNewPage:=0;
		END_IF;
		T_Visu.T_PlcParam.dwActualPage:=0;
		T_Visu.T_PlcParam.dwPreviousPage:=0;
		T_Visu.ptrT_ExchgParam^.T_Visu.iQVisActivNewPage:=0;
		wNormalLayerActivTask:=1;
		wSpecialLayerGeneralActivTask:=1;
		wSpecialLayerToolRotActivTask:=1;
		wSpecialLayerWireFeedActivTask:=1;
		wSpecialLayerGrindAxisActivTask:=1;
		wNormalLayerActivPage:=10;
		wSpecialLayerGeneralActivPage:=110;
		wSpecialLayerToolRotActivPage:=210;
		wSpecialLayerWireFeedActivPage:=310;
		wSpecialLayerGrindAxisActivPage:=410;
		wTmpNormalLayerActivTask:=1;
		wTmpSpecialLayerGeneralActivTask:=1;
		wTmpSpecialLayerToolRotActivTask:=1;
		wTmpSpecialLayerWireFeedActivTask:=1;
		wTmpSpecialLayerGrindAxisActivTask:=1;
		T_Visu.ptrT_ExchgParam^.T_TouchScreenNavPanel.wState:=1;
		T_Visu.ptrT_ExchgParam^.T_Visu.bActivSpecialLayer:=0;
		T_Visu.ptrT_ExchgParam^.T_TouchScreenBtPanel.iStateBtLeft:=0;
		wStandardPageNr:=10;
		T_Visu.ptrT_ExchgParam^.T_Visu.T_Level.iPwSystem:=999;
		FOR ii:=1 TO 6 DO
			awNormalLayerActivPage[ii]:=wStandardPageNr;
			wStandardPageNr:=wStandardPageNr + 10;
		END_FOR;
		wStandardPageNr:=110;
		FOR ii:=1 TO 6 DO
			awSpecialLayerGeneralActivPage[ii]:=wStandardPageNr;
			wStandardPageNr:=wStandardPageNr + 10;
		END_FOR;
		wStandardPageNr:=210;
		FOR ii:=1 TO 6 DO
			awSpecialLayerToolRotActivPage[ii]:=wStandardPageNr;
			wStandardPageNr:=wStandardPageNr + 10;
		END_FOR;
		wStandardPageNr:=310;
		FOR ii:=1 TO 6 DO
			awSpecialLayerWireFeedActivPage[ii]:=wStandardPageNr;
			wStandardPageNr:=wStandardPageNr + 10;
		END_FOR;
		wStandardPageNr:=410;
		FOR ii:=1 TO 6 DO
			awSpecialLayerGrindAxisActivPage[ii]:=wStandardPageNr;
			wStandardPageNr:=wStandardPageNr + 10;
		END_FOR;
		(* Activ reset structure control action *)
		T_Visu.T_CtrleAction.xReset:=TRUE;
		(* Activ reset structure control process *)
		T_Visu.T_CtrleProcess.xReset:=TRUE;
		(* Init. pw value *)
		T_Visu.ptrT_ExchgParam^.T_Visu.T_Level.iPwSystem:=999;
		(* Init. Error *)
		T_Visu.ptrT_ExchgParam^.T_Visu.T_Message.iState:=0;
		T_Visu.ptrT_ExchgParam^.T_Visu.T_Message.sDynamicTextEnglish:='';
		T_Visu.ptrT_ExchgParam^.T_Visu.T_Message.sDynamicTextDeutsch:='';
		T_Visu.ptrT_ExchgParam^.T_Visu.T_Message.sDynamicTextFrancais:='';
		T_Visu.ptrT_ExchgParam^.T_TouchScreenBtPanel.iStateBtLeft:=0;
		T_Visu.ptrT_ExchgParam^.T_Cylinder.iSelectCylinder_Sonder1:=1;
		T_Visu.ptrT_ExchgParam^.T_StationCommon.iWireFeederAngleRefIndex:=0;
		T_Visu.ptrT_ExchgParam^.T_TeachIn.iSelectAxisGrind:=1;
		T_Visu.ptrT_ExchgParam^.T_TeachIn.iSelectAxisToolRotation:=1;
		T_Visu.ptrT_ExchgParam^.T_TeachIn.iSelectAxisWireFeeder:=1;
		T_Visu.ptrT_ExchgParam^.T_TeachIn.xSlowFastToolRotation:=FALSE;
		T_Visu.ptrT_ExchgParam^.T_TeachIn.xSlowFastToolFeed:=FALSE;
		T_Visu.ptrT_ExchgParam^.T_TeachIn.xSlowFastGrindFeeder:=FALSE;
		T_Visu.ptrT_ExchgParam^.T_InfoValueCommon.rToolTensionForce:=T_NovRAM.T_Data.T_ProcessImageData.T_ProcessPara.rToolTensionProcess;
		(* active confirmation *)
		xConfirmResetFB:=TRUE;
		(* exit function bloc *)
		RETURN;
	ELSE
		IF xConfirmResetFB THEN
			(* confirm reset FB *)
			T_Visu.T_CtrleVisu.xDone:=TRUE;
			T_Visu.T_CtrleVisu.xErr:=FALSE;
			T_Visu.T_CtrleVisu.udiErrorID:=0;
			(* reset variable *)
			xConfirmResetFB:=FALSE;
			(* activ research if Qvis is activ *)
			xQvisActiv:=TRUE;
			T_Visu.T_CtrleVisu.xQvis:=FALSE;
			dwInCount_QVisCmd:=T_CtrleQVis.dwInCount;
		END_IF
	END_IF

(* determin if qvis activ *)
	IF xQvisActiv THEN
		(* timer time off  *)
		TimerQVis(IN:=TRUE,PT:=T#2s);
		IF dwInCount_QVisCmd = T_CtrleQVis.dwInCount THEN
			(* Init. command *)
			T_CtrleQVis.dwInCommand:=1;
			T_CtrleQVis.dwInQVisCtrlAddress:=ADR(T_CtrleQVis);
			T_CtrleQVis.dwInParameterAddress:=ADR(T_Visu.T_PlcParam.dwSetNewPage);
			(* start command *)
			T_CtrleQVis.dwInCount:=T_CtrleQVis.dwInCount+1;
			(* Activ Timer *)
			TimerQVis(IN:=FALSE);
		ELSE
			IF T_CtrleQVis.dwInCount = T_CtrleQVis.dwOutCount THEN
			(* command done *)
				IF T_CtrleQVis.diOutStatus = 0 THEN
				(* command done without error *)
					xQvisActiv:=FALSE;
					T_Visu.T_CtrleVisu.xQvis:=TRUE;
					T_Visu.T_PlcParam.dwActualPage:=T_Visu.T_PlcParam.dwSetNewPage;
				END_IF
			ELSE
			(* test time off, restart command *)
				IF TimerQVis.Q THEN
					dwInCount_QVisCmd:=T_CtrleQVis.dwInCount;
				END_IF
			END_IF
		END_IF
	END_IF

(* exit FB if Qvis inactiv *)
	IF NOT(T_Visu.T_CtrleVisu.xQvis) THEN RETURN; END_IF

	IF (T_Visu.T_PlcParam.dwActualPage > 0) AND (T_Visu.T_PlcParam.dwActualPage <= 999) THEN
		(* copy config page structure *)
		T_ConfigPage:=T_Visu.T_ConfigPage[T_Visu.T_PageIndex[T_Visu.T_PlcParam.dwActualPage].iIndexConfigPage];
		T_Visu.ptrT_ExchgParam^. T_TouchScreenNavPanel.wNotMasktext:=T_ConfigPage.wMaskTouchScreenNavPanel;
		T_Visu.ptrT_ExchgParam^.T_TouchScreenBtPanel.iNotMaskTextBt:=16#0;
		T_Visu.ptrT_ExchgParam^.T_TouchScreenBtPanel.iNotMaskTextBt:=WORD_TO_INT(INT_TO_WORD(T_Visu.ptrT_ExchgParam^.T_TouchScreenBtPanel.iNotMaskTextBt) OR T_ConfigPage.wMaskBtPanelRight);
		T_Visu.ptrT_ExchgParam^.T_TouchScreenBtPanel.iNotMaskTextBt:=WORD_TO_INT(INT_TO_WORD(T_Visu.ptrT_ExchgParam^.T_TouchScreenBtPanel.iNotMaskTextBt) OR T_ConfigPage.wMaskBtPanelLeft);
		T_Visu.ptrT_ExchgParam^.T_TouchScreenBtPanel.iNotMaskTextBt:=WORD_TO_INT(NOT(INT_TO_WORD(T_Visu.ptrT_ExchgParam^.T_TouchScreenBtPanel.iNotMaskTextBt)));
	END_IF;

(* monitor page Errorlist for Machine *)
	xTmp:=	(T_Visu.T_PlcParam.dwActualPage = 60) OR
			(T_Visu.T_PlcParam.dwActualPage = 160) OR
			(T_Visu.T_PlcParam.dwActualPage = 260) OR
			(T_Visu.T_PlcParam.dwActualPage = 360) OR
			(T_Visu.T_PlcParam.dwActualPage = 460);
	IF xTmp THEN
		(* Check if Station will be changed without changing the Error Page *)
		IF (dwTmpActualPage <> T_Visu.T_PlcParam.dwActualPage) THEN
			xUpdateErrorList:=TRUE;
			dwTmpActualPage:=T_Visu.T_PlcParam.dwActualPage;
		END_IF;
	END_IF;
	IF xTmp OR xUpdateErrorList THEN
		IF NOT(xTmp) AND xUpdateErrorList THEN
			RisingEdgeErrorList(CLK:=xUpdateErrorList);
		ELSE
			RisingEdgeErrorList(CLK:=xTmp AND NOT(xUpdateErrorList));
		END_IF;
		xUpdateErrorList:=FALSE;
		IF RisingEdgeErrorList.Q THEN
			FBQVisErrorList(	T_ErrorList:= T_ErrorList,
							T_ErrorNrList:= T_NovRAM.T_Data.T_ErrorNrList,
							T_MsgErrorEnglish:= T_Visu.ptrT_ExchgParam^.T_Visu.T_MsgErrorEnglish,
							T_MsgErrorDeutsch:= T_Visu.ptrT_ExchgParam^.T_Visu.T_MsgErrorDeutsch,
							T_MsgErrorFrancais:= T_Visu.ptrT_ExchgParam^.T_Visu.T_MsgErrorFrancais);
		END_IF;
	ELSE
		RisingEdgeErrorList(CLK:=FALSE);
	END_IF;

(* Refresh Errorlist for Machine and Station *)
	FBSetErrorList(	TControlStation:= T_Station.TControl,
					TProcess:= T_Process,
					xParameterSaved:= xParameterSavedErrorList,
					T_ErrorNrList:= T_NovRAM.T_Data.T_ErrorNrList,
					xSetForceError:= T_Visu.ptrT_ExchgParam^.T_SafetyCtrl.xSetForceError,
					diSetForceErrorNr:= T_Visu.ptrT_ExchgParam^.T_SafetyCtrl.diSetForceErrorNr);
	IF FBSetErrorList.xSaveParameter THEN
		IF T_Visu.T_CtrleAction.xDone AND NOT(T_Visu.T_CtrleAction.xExecute) AND T_NovRAM.T_Ctrle.xDone AND NOT(T_NovRAM.T_Ctrle.xExecute) THEN
			xParameterSavedErrorList:=TRUE;
			xUpdateErrorList:=TRUE;
			T_NovRAM.T_Ctrle.xExecute:=TRUE;
			T_NovRAM.T_Ctrle.iFunction:=2;
			T_NovRAM.T_Data.T_ErrorNrList;
		END_IF;
	END_IF;

(* Monitoring Visu Parameter *)
	T_Visu.ptrT_ExchgParam^.T_StationCommon.rConvertMaxToolLength:=T_NovRAM.T_Data.T_Standard.T_MachineConfig.rConfigMaxToolLength * 10.0;	(* convert from cm to mm *)
	T_Visu.ptrT_ExchgParam^.T_StationCommon.T_ParamToolTensionSystem.rMaxForceTT:=T_NovRAM.T_Data.T_Standard.T_ToolTensionSystem.rMaxForceTT;
	IF (T_NovRam.T_Data.T_Standard.T_MachineConfig.iConfigMachineType = 2) THEN
		xMicroRodActive:=TRUE;
	ELSE
		xMicroRodActive:=FALSE;
	END_IF;
	IF (T_Visu.T_PlcParam.dwActualPage = 170) AND ((T_Visu.ptrT_ExchgParam^.T_Config.iEditParam >= 120) AND (T_Visu.ptrT_ExchgParam^.T_Config.iEditParam <= 129)) THEN
		IF NOT(xFirstReadParaList) THEN
			iTmpSelectParaList:=T_Visu.ptrT_ExchgParam^.T_Config.iSelectParaList;
		END_IF;
		xFirstReadParaList:=TRUE;
		T_Visu.ptrT_ExchgParam^.T_Config.xBlockParaListNavi:=FALSE;
		T_Visu.ptrT_ExchgParam^.T_Config.xBlockParaListNavi1:=TRUE;
		T_Visu.ptrT_ExchgParam^.T_Config.xBlockProfilList:=FALSE;
		T_Visu.ptrT_ExchgParam^.T_Config.xBlockNavParaList:=FALSE;
		T_Visu.ptrT_ExchgParam^.T_Config.iEditParam:=iFctGetEditParaList(	dwActualPage:=120,
																	xMicroRodActive:=xMicroRodActive,
																	iSelectParaList:=T_Visu.ptrT_ExchgParam^.T_Config.iSelectParaList,
																	iSelectParaListTeachRot:=T_Visu.ptrT_ExchgParam^.T_Config.iSelectParaListTeachRot);
		(* 09.12.2010 KFS:	{	*)
		IF (T_ExchgParam.T_Visu.T_Level.iActLevel <>2) THEN
			IF  (T_Visu.ptrT_ExchgParam^.T_Config.iEditParam = 121) THEN
				 T_Visu.ptrT_ExchgParam^.T_Config.iEditParam:= 126;
			ELSIF ( T_Visu.ptrT_ExchgParam^.T_Config.iEditParam = 123) THEN
				 T_Visu.ptrT_ExchgParam^.T_Config.iEditParam:= 127;
			ELSIF ( T_Visu.ptrT_ExchgParam^.T_Config.iEditParam = 125) THEN
				 T_Visu.ptrT_ExchgParam^.T_Config.iEditParam:= 128;
			END_IF;
		END_IF;
		(* 09.12.2010 KFS:	}	*)
		IF (iTmpSelectParaList <> T_Visu.ptrT_ExchgParam^.T_Config.iSelectParaList) THEN
			iTmpSelectParaList:=T_Visu.ptrT_ExchgParam^.T_Config.iSelectParaList;
			xResetParaListValue:=TRUE;
		END_IF;
	ELSE
		xFirstReadParaList:=FALSE;
		T_Visu.ptrT_ExchgParam^.T_Config.xBlockNavParaList:=TRUE;
	END_IF;
	IF (T_Visu.T_PlcParam.dwActualPage = 270) AND ((T_Visu.ptrT_ExchgParam^.T_Config.iEditParam >= 210) AND (T_Visu.ptrT_ExchgParam^.T_Config.iEditParam <= 219)) THEN
		IF NOT(xFirstReadParaList1) THEN
			iTmpSelectParaList1:=T_Visu.ptrT_ExchgParam^.T_Config.iSelectParaListTeachRot;
		END_IF;
		xFirstReadParaList1:=TRUE;
		T_Visu.ptrT_ExchgParam^.T_Config.xBlockNavParaListTeachRot:=FALSE;
		T_Visu.ptrT_ExchgParam^.T_Config.iEditParam:=iFctGetEditParaList(	dwActualPage:=210,
																	xMicroRodActive:=xMicroRodActive,
																	iSelectParaList:=T_Visu.ptrT_ExchgParam^.T_Config.iSelectParaListTeachRot,
																	iSelectParaListTeachRot:=T_Visu.ptrT_ExchgParam^.T_Config.iSelectParaListTeachRot);
		IF (iTmpSelectParaList1 <> T_Visu.ptrT_ExchgParam^.T_Config.iSelectParaListTeachRot) THEN
			iTmpSelectParaList1:=T_Visu.ptrT_ExchgParam^.T_Config.iSelectParaListTeachRot;
			xResetParaListValue:=TRUE;
		END_IF;
	ELSE
		xFirstReadParaList1:=FALSE;
		T_Visu.ptrT_ExchgParam^.T_Config.xBlockNavParaListTeachRot:=TRUE;
	END_IF;
	xTmp:=	(T_Visu.T_PlcParam.dwActualPage = 170) OR
			(T_Visu.T_PlcParam.dwActualPage = 270) OR
			(T_Visu.T_PlcParam.dwActualPage = 370) OR
			(T_Visu.T_PlcParam.dwActualPage = 470);
	IF xTmp AND (T_Visu.ptrT_ExchgParam^.T_Config.iEditParam = 0) THEN
		T_Visu.ptrT_ExchgParam^.T_Config.xBlockParaListNavi:=TRUE;
		T_Visu.ptrT_ExchgParam^.T_Config.xBlockParaListNavi1:=TRUE;
	END_IF;

(* Monitor dynamic mask for button panel left and right and function panel *)
	IF T_Visu.T_CtrleProcess.xDone OR T_Visu.T_CtrleProcess.xErr THEN
	(* Set the standard mask *)
		wMaskBtPanelLeft:=T_ConfigPage.wMaskBtPanelLeft;
		wMaskBtPanelRight:=T_ConfigPage.wMaskBtPanelRight;
		wMaskFunctionPanel:=T_ConfigPage.wMaskFunctionPanel;
	(* Set the dynamic mask *)
	ELSE	wMaskBtPanelLeft:=T_ConfigPage.wMaskBtPanelLeft AND T_ConfigPage.wMaskActiveMachineBtPanelLeft;
			wMaskBtPanelRight:=T_ConfigPage.wMaskActiveMachineBtPanelRight;
			wMaskFunctionPanel:=T_ConfigPage.wMaskActiveMachineFunctionPanel;
	END_IF
	(* Check activ Page *)
	IF (T_Visu.T_PlcParam.dwActualPage = 170) OR (T_Visu.T_PlcParam.dwActualPage = 270) OR (T_Visu.T_PlcParam.dwActualPage = 370) OR (T_Visu.T_PlcParam.dwActualPage = 470) THEN
		IF (T_Visu.ptrT_ExchgParam^.T_Config.iEditParam = 0) THEN
			wMaskBtPanelRight:=16#0;
		END_IF;
		IF (T_Visu.ptrT_ExchgParam^.T_Config.iEditParam = 130) OR (T_Visu.ptrT_ExchgParam^.T_Config.iEditParam = 131) THEN
			wMaskBtPanelRight:=16#0;
		END_IF;
	END_IF;
	(* Config. divers mask *)
	T_Visu.ptrT_ExchgParam^.T_TouchScreenBtPanel.iNotMaskTextBt
	 :=(16#1F XOR wMaskBtPanelLeft) OR (16#3E0 XOR wMaskBtPanelRight);
	(* management Fn button panel availability *)
	T_Visu.ptrT_ExchgParam^.T_BtFunctionPanel.wNotMasktext:=16#FFF XOR wMaskFunctionPanel;
	(* management navigation panel mask *)
	T_Visu.ptrT_ExchgParam^.T_TouchScreenNavPanel.wNotMasktext:=T_ConfigPage.wMaskTouchScreenNavPanel;


MaskFunctionButton;

(************************************************************************************************************************************************************************)
(********start of the managment of the external start-stop button, special button and function button and task button and external tool buttons********)
(************************************************************************************************************************************************************************)
CtrlStartStopButton;
CtrlPanelLeftButton;
CtrlPanelRightButton;
CtrlFunctionButton;
CtrlTaskBar;
(************************************************************************************************************************************************************************)
(*********end of the managment of the external start-stop button, special button and function button and task button and external tool buttons********)
(************************************************************************************************************************************************************************)



(* set system level *)
	IF (T_Visu.ptrT_ExchgParam^.T_Visu.T_Level.iPwSystem <> 999) AND (T_Visu.T_PlcParam.dwActualPage = 40) THEN
		IF T_Visu.ptrT_ExchgParam^.T_Visu.T_Level.iPwSystem = iPwSystem THEN
		(* pw correct *)
			T_Visu.ptrT_ExchgParam^.T_Visu.T_Level.iActLevel:=2;
			T_Visu.ptrT_ExchgParam^.T_Visu.T_Message.iState:=2;
		(* wrong pw *)
		ELSE 	T_Visu.ptrT_ExchgParam^.T_Visu.T_Message.iState:=3; END_IF
		T_Visu.ptrT_ExchgParam^.T_Visu.T_Level.iPwSystem:=999;
	END_IF
	IF (T_Visu.T_PlcParam.dwActualPage = 40) THEN
		RisingEdgeDynPassword(CLK:=TRUE);
		IF RisingEdgeDynPassword.Q THEN
			fbGetCpuAccount;
			fbPwSystem(	dwCounter:=fbGetCpuAccount.fbGetCpuCounter.dwCpuCntHi+fbGetCpuAccount.fbGetCpuCounter.dwCpuCntLo,
						iRandom=>T_Visu.ptrT_ExchgParam^.T_Visu.T_Level.iRandom,
						iPwSystem=>iPwSystem);
		END_IF;
	ELSE
		RisingEdgeDynPassword(CLK:=FALSE);
	END_IF;

(************************************************************************************************************************************************************************)
(**********************************						Profile Management Start						****************************************)
(************************************************************************************************************************************************************************)

(* Update profile list *)
	IF xUpdateProfileList THEN
		xTmp:= 	iPointerListProfile > 0
				AND (iPointerListProfile+4) <= csiMaxProfile;
		IF xTmp THEN
			jj:=1;
			FOR ii:=iPointerListProfile TO iPointerListProfile+4 DO
				T_Visu.ptrT_ExchgParam^.T_ProfileCommon.T_ProfileList[jj].iNumber:=ii;
				T_Visu.ptrT_ExchgParam^.T_ProfileCommon.T_ProfileList[jj].sName:=T_NovRam.T_Data.T_IDProfileStation[ii].sName;
				jj:=jj+1;
			END_FOR
		END_IF
		(* confirm update *)
		xUpdateProfileList:=FALSE;
	END_IF

(* Compare Profile and Process value *)
	xTmp:=	(T_Visu.ptrT_ExchgParam^.T_StationCommon.T_InfoProcess.iProfile <> 0);
	IF xTmp THEN
		fbCompareProfileProcessValue(T_Data_ProcessImageLoadData:=T_NovRam.T_Data.T_ProcessImageLoadData,
									T_Data_ProcessImageData:=T_NovRam.T_Data.T_ProcessImageData,
									xMicroRodActive:=xMicroRodActive);
		T_Visu.ptrT_ExchgParam^.T_StationCommon.T_InfoProcess.xOnlineValueModified:=fbCompareProfileProcessValue.xProcessValueModified;
	END_IF

(* monitor change actual profile common *)
	IF (T_Visu.T_PlcParam.dwActualPage = 130) THEN
		IF T_Visu.ptrT_ExchgParam^.T_ProfileCommon.T_Id.iNumber<>iActualActiveProfile THEN
			IF T_Visu.T_CtrleAction.xDone THEN
				(* set value from selected profile *)
				T_Visu.ptrT_ExchgParam^.T_ProfileCommon.T_Id.sName
					:=T_NovRam.T_Data.T_IDProfileStation[T_Visu.ptrT_ExchgParam^.T_ProfileCommon.T_Id.iNumber].sName;
				(* save value from selected profile *)
				iActualActiveProfile:=T_Visu.ptrT_ExchgParam^.T_ProfileCommon.T_Id.iNumber;
			END_IF
		END_IF
	END_IF

(* Pointer Profile List Up/Down Slow *)
	RisingEdgePtrProfileListUpDown(CLK:=	T_Visu.ptrT_ExchgParam^.T_ProfileCommon.T_ProfileManage.xListProfileUp
										OR T_Visu.ptrT_ExchgParam^.T_ProfileCommon.T_ProfileManage.xListProfileDown);
	IF RisingEdgePtrProfileListUpDown.Q THEN
		IF T_Visu.ptrT_ExchgParam^.T_ProfileCommon.T_ProfileManage.xListProfileUp THEN
			iPointerListProfile:=iPointerListProfile-5;
		ELSE iPointerListProfile:=iPointerListProfile+5; END_IF
		(* min/max=1/6 *)
		IF iPointerListProfile>(csiMaxProfile -5) THEN iPointerListProfile:=(csiMaxProfile - 4); END_IF
		IF iPointerListProfile<0 THEN iPointerListProfile:=1; END_IF
		T_Visu.ptrT_ExchgParam^.T_ProfileCommon.T_ProfileManage.xListProfileUp:=FALSE;
		T_Visu.ptrT_ExchgParam^.T_ProfileCommon.T_ProfileManage.xListProfileDown:=FALSE;
		(* Update display  list *)
		xUpdateProfileList:=TRUE;
	END_IF

(* Pointer Profile List Up/Down Fast *)
	RisingEdgePtrProfileListUpDown(CLK:=	T_Visu.ptrT_ExchgParam^.T_ProfileCommon.T_ProfileManage.xListProfileUpFast
										OR T_Visu.ptrT_ExchgParam^.T_ProfileCommon.T_ProfileManage.xListProfileDownFast);
	IF RisingEdgePtrProfileListUpDown.Q THEN
		IF T_Visu.ptrT_ExchgParam^.T_ProfileCommon.T_ProfileManage.xListProfileUpFast THEN
			iPointerListProfile:=iPointerListProfile-10;
		ELSE iPointerListProfile:=iPointerListProfile+10; END_IF
		(* min/max=1/6 *)
		IF iPointerListProfile>(csiMaxProfile -5) THEN iPointerListProfile:=(csiMaxProfile - 4); END_IF
		IF iPointerListProfile<0 THEN iPointerListProfile:=1; END_IF
		T_Visu.ptrT_ExchgParam^.T_ProfileCommon.T_ProfileManage.xListProfileUpFast:=FALSE;
		T_Visu.ptrT_ExchgParam^.T_ProfileCommon.T_ProfileManage.xListProfileDownFast:=FALSE;
		(* Update display  list *)
		xUpdateProfileList:=TRUE;
	END_IF

(************************************************************************************************************************************************************************)
(**********************************						Profile Management End						****************************************)
(************************************************************************************************************************************************************************)

(* Display info or warning message *)
	RisingEdgeKeySwitch1(CLK:=xSecurityKey);
	FailingEdgeKeySwitch1(CLK:=xSecurityKey);
	IF T_Visu.ptrT_ExchgParam^.T_Visu.T_Message.iState <> 0 THEN
		(* info message *)
		IF T_Visu.ptrT_ExchgParam^.T_Visu.T_Message.iState < 100THEN
		(* activ message during 3s, after that the message will be cleared *)
			TimerDisplayMessage(IN:=TRUE,PT:=T#3s);
			IF TimerDisplayMessage.Q THEN
				T_Visu.ptrT_ExchgParam^.T_Visu.T_Message.iState:=0;
					T_ExchgParam.T_FunctionCommon.xWarmUp_MessageWarning_2:=FALSE;   (* SOA 20.02.2023 *)
				TimerDisplayMessage(IN:=FALSE);
			END_IF
			IF (T_Visu.ptrT_ExchgParam^.T_Visu.T_Message.iState = 2) THEN
				IF (TimerDisplayMessage.ET > T#0.5s) THEN
					T_Visu.ptrT_ExchgParam^.T_Visu.T_Message.iState:=0;
						T_ExchgParam.T_FunctionCommon.xWarmUp_MessageWarning_2:=FALSE;
					TimerDisplayMessage(IN:=FALSE);
				END_IF;
			END_IF;
		(* disable timer *)
		ELSE TimerDisplayMessage(IN:=FALSE); END_IF

		(* warning message *)
		xTmp:=	(T_Visu.ptrT_ExchgParam^.T_Visu.T_Message.iState > 100 AND T_Visu.ptrT_ExchgParam^.T_Visu.T_Message.iState <200)
				AND T_Visu.T_CtrleAction.xDone;
		RisingEdgeReleaseWarning(CLK:=wActivBtLeft <> 16#0 OR T_Visu.ptrT_ExchgParam^.T_BtFunctionPanel.wActivBt <> 16#0);
		(* the warning will be cleared by the operator *)
		IF xTmp AND (RisingEdgeReleaseWarning.Q OR RisingEdgeKeySwitch1.Q OR FailingEdgeKeySwitch1.Q) THEN
			IF (T_Visu.ptrT_ExchgParam^.T_Visu.T_Message.iState <> 120) THEN
				T_Visu.ptrT_ExchgParam^.T_Visu.T_Message.iState:=0;
			END_IF;
		END_IF
	END_IF

(* Monitor dynamic error text *)
	xTmp:=	T_Visu.ptrT_ExchgParam^.T_Visu.T_Message.sDynamicTextEnglish <> ''
			AND T_Visu.ptrT_ExchgParam^.T_Visu.T_Message.iState <> 401;
	IF xTmp THEN
		bStateMachine:=0;
		T_Visu.ptrT_ExchgParam^.T_Visu.T_Message.iState:=401;
		xSetStateMachine:=TRUE;
		xCheckQuitError:=TRUE;
	END_IF
	IF xCheckQuitError THEN
		IF (T_Visu.ptrT_ExchgParam^.T_Visu.T_Message.iState <> 401) THEN
			xSetStateMachine:=TRUE;
			xCheckQuitError:=FALSE;
			IF NOT(T_TwinSafeOut.QxContactor_K3) OR NOT(T_TwinSafeOut.QxContactor_K4) THEN
				bStateMachine:=3;
			ELSE
				bStateMachine:=1;
			END_IF;
		END_IF;
	END_IF;
	IF NOT(T_TwinSafeIn.IxPowerSupplyEcoStep) THEN
		bStateMachine:=4;
	END_IF;
	IF xSetStateMachine THEN
		xSetStateMachine:=FALSE;
		T_Visu.ptrT_ExchgParam^.T_SafetyCtrl.bStateAutoGeometry:=bStateMachine;
		T_Visu.ptrT_ExchgParam^.T_SafetyCtrl.bStateAutoGroove:=bStateMachine;
		T_Visu.ptrT_ExchgParam^.T_SafetyCtrl.bStateReference:=bStateMachine;
		T_Visu.ptrT_ExchgParam^.T_SafetyCtrl.bStateToolCalibration:=bStateMachine;
		T_Visu.ptrT_ExchgParam^.T_SafetyCtrl.bStateToolTorque:=bStateMachine;
		T_Visu.ptrT_ExchgParam^.T_SafetyCtrl.bStateTeachInToolLeft:=bStateMachine;
		T_Visu.ptrT_ExchgParam^.T_SafetyCtrl.bStateTeachInToolCenter:=bStateMachine;
		T_Visu.ptrT_ExchgParam^.T_SafetyCtrl.bStateTeachInToolRight:=bStateMachine;
		T_Visu.ptrT_ExchgParam^.T_SafetyCtrl.bStateTeachInToolFeeder:=bStateMachine;
		T_Visu.ptrT_ExchgParam^.T_SafetyCtrl.bStateReferenceMaxToolLength:=bStateMachine;
		T_Visu.ptrT_ExchgParam^.T_SafetyCtrl.bStateTeachInGrindFeeder:=bStateMachine;
		T_Visu.ptrT_ExchgParam^.T_StationCommon.iWireFeederRefIndexState:=BYTE_TO_INT(bStateMachine);
	END_IF;

(* Reset settled value on the parameter list, without saved *)
	IF xResetParaListValue OR T_Visu.T_CtrleAction.xResetParaListValue THEN
		T_Visu.T_CtrleAction.xResetParaListValue:=FALSE;
		xResetParaListValue:=FALSE;
		T_Visu.ptrT_ExchgParam^.T_TeachIn.TParam_ToolLeft:=T_NovRAM.T_Data.T_Standard.T_TeachINToolLeft;
		T_Visu.ptrT_ExchgParam^.T_TeachIn.TParam_ToolCenter:=T_NovRAM.T_Data.T_Standard.T_TeachINToolCenter;
		T_Visu.ptrT_ExchgParam^.T_TeachIn.TParam_ToolRight:=T_NovRAM.T_Data.T_Standard.T_TeachINToolRight;
		T_Visu.ptrT_ExchgParam^.T_TeachIn.TParam_ToolFeeder:=T_NovRAM.T_Data.T_Standard.T_TeachINToolFeeder;
		T_Visu.ptrT_ExchgParam^.T_TeachIn.TParam_GrindFeeder:=T_NovRAM.T_Data.T_Standard.T_TeachINGrindFeeder;
		T_Visu.ptrT_ExchgParam^.T_TeachIn.TParam_AxisPosition:=T_NovRAM.T_Data.T_Standard.T_AxisPosition;
		T_Visu.ptrT_ExchgParam^.T_StationCommon.iConfigMachineType:=T_NovRAM.T_Data.T_Standard.T_MachineConfig.iConfigMachineType;
		T_Visu.ptrT_ExchgParam^.T_StationCommon.iConfigAxisType:=T_NovRAM.T_Data.T_Standard.T_MachineConfig.iConfigAxisType;
		T_Visu.ptrT_ExchgParam^.T_StationCommon.iConfigVisuNavigation:=T_NovRAM.T_Data.T_Standard.T_MachineConfig.iConfigVisuNavigation;
		T_Visu.ptrT_ExchgParam^.T_StationCommon.rConfigMaxToolLength:=T_NovRAM.T_Data.T_Standard.T_MachineConfig.rConfigMaxToolLength;
		T_Visu.ptrT_ExchgParam^.T_StationCommon.T_ParamToolTensionSystem:=T_NovRAM.T_Data.T_Standard.T_ToolTensionSystem;
		T_Visu.ptrT_ExchgParam^.T_Cylinder.T_ParamToolTension:=T_NovRAM.T_Data.T_Standard.T_Cyl_ToolTension;
		T_Visu.ptrT_ExchgParam^.T_StationCommon.T_AutoGeometryPara:=T_NovRAM.T_Data.T_ProcessImageData.T_AutoGeometryPara;
		T_Visu.ptrT_ExchgParam^.T_StationCommon.T_AutoGroovePara:=T_NovRAM.T_Data.T_ProcessImageData.T_AutoGroovePara;
		T_Visu.ptrT_ExchgParam^.T_StationCommon.T_CalibrationPara:=T_NovRAM.T_Data.T_ProcessImageData.T_CalibrationPara;
		T_Visu.ptrT_ExchgParam^.T_StationCommon.T_ProcessPara:=T_NovRAM.T_Data.T_ProcessImageData.T_ProcessPara;
		T_Visu.ptrT_ExchgParam^.T_StationCommon.T_InfoProcess.iProfile:=T_Visu.ptrT_ExchgParam^.T_ProfileCommon.T_Id.iNumber;
		T_Visu.ptrT_ExchgParam^.T_StationCommon.T_InfoProcess.sProfileName:=T_NovRam.T_Data.T_IDProfileStation[T_Visu.ptrT_ExchgParam^.T_ProfileCommon.T_Id.iNumber].sName;
		T_Visu.ptrT_ExchgParam^.T_GeometryCommon.T_Geometry:=T_NovRAM.T_Data.T_ProcessImageData.T_GeometryPara;
		T_Visu.ptrT_ExchgParam^.T_StationCommon.T_PrismPara:=T_NovRAM.T_Data.T_ProcessImageData.T_PrismPara;
		T_Visu.ptrT_ExchgParam^.T_GeometryCommon.rMinToolDiameter:=T_NovRAM.T_Data.T_ProcessImageData.T_PrismPara.rToolDiameterMin;
		T_Visu.ptrT_ExchgParam^.T_GeometryCommon.rMaxToolDiameter:=T_NovRAM.T_Data.T_ProcessImageData.T_PrismPara.rToolDiameterMax;
		T_Visu.ptrT_ExchgParam^.T_GeometryCommon.rMinToolLength:=0.1;
		T_Visu.ptrT_ExchgParam^.T_GeometryCommon.rMaxToolLength:=T_NovRAM.T_Data.T_Standard.T_MachineConfig.rConfigMaxToolLength;
		T_Visu.ptrT_ExchgParam^.T_StationCommon.rConfigMaxToolLengthOriginal:=T_NovRAM.T_Data.T_Standard.T_MachineConfig.rConfigMaxToolLengthOriginal;
	END_IF;

(* Monitoring Process value *)
	IF T_Process.xReferenced THEN T_Visu.ptrT_ExchgParam^.T_Machine.T_Process.wState:=T_Visu.ptrT_ExchgParam^.T_Machine.T_Process.wState OR 16#1;
		ELSE T_Visu.ptrT_ExchgParam^.T_Machine.T_Process.wState:=T_Visu.ptrT_ExchgParam^.T_Machine.T_Process.wState AND 16#FE; END_IF
	IF NOT(T_Process.xEnd) THEN T_Visu.ptrT_ExchgParam^.T_Machine.T_Process.wState:=T_Visu.ptrT_ExchgParam^.T_Machine.T_Process.wState OR 16#2;
		ELSE T_Visu.ptrT_ExchgParam^.T_Machine.T_Process.wState:=T_Visu.ptrT_ExchgParam^.T_Machine.T_Process.wState AND 16#FD; END_IF
	IF T_Process.xError THEN T_Visu.ptrT_ExchgParam^.T_Machine.T_Process.wState:=T_Visu.ptrT_ExchgParam^.T_Machine.T_Process.wState OR 16#4;
		ELSE T_Visu.ptrT_ExchgParam^.T_Machine.T_Process.wState:=T_Visu.ptrT_ExchgParam^.T_Machine.T_Process.wState AND 16#FB; END_IF
	IF T_Process.xRdy THEN T_Visu.ptrT_ExchgParam^.T_Machine.T_Process.wState:=T_Visu.ptrT_ExchgParam^.T_Machine.T_Process.wState OR 16#8;
		ELSE T_Visu.ptrT_ExchgParam^.T_Machine.T_Process.wState:=T_Visu.ptrT_ExchgParam^.T_Machine.T_Process.wState AND 16#F7; END_IF
	IF T_Process.xEnd THEN T_Visu.ptrT_ExchgParam^.T_Machine.T_Process.wState:=T_Visu.ptrT_ExchgParam^.T_Machine.T_Process.wState OR 16#10;
		ELSE T_Visu.ptrT_ExchgParam^.T_Machine.T_Process.wState:=T_Visu.ptrT_ExchgParam^.T_Machine.T_Process.wState AND 16#EF; END_IF
	IF T_Process.xProcessHold THEN T_Visu.ptrT_ExchgParam^.T_Machine.T_Process.wState:=T_Visu.ptrT_ExchgParam^.T_Machine.T_Process.wState OR 16#40;
		ELSE T_Visu.ptrT_ExchgParam^.T_Machine.T_Process.wState:=T_Visu.ptrT_ExchgParam^.T_Machine.T_Process.wState AND 16#BF; END_IF
	IF T_Process.xStop THEN T_Visu.ptrT_ExchgParam^.T_Machine.T_Process.wState:=T_Visu.ptrT_ExchgParam^.T_Machine.T_Process.wState OR 16#80;
		ELSE T_Visu.ptrT_ExchgParam^.T_Machine.T_Process.wState:=T_Visu.ptrT_ExchgParam^.T_Machine.T_Process.wState AND 16#7F; END_IF

(* Monitoring Station value *)
	IF T_Station.TControl.xEnd AND T_Station.TControl.xRdy AND T_Station.TControl.xEnable THEN
		T_Visu.ptrT_ExchgParam^.T_StationCommon.bStateMachine:=T_Visu.ptrT_ExchgParam^.T_StationCommon.bStateMachine OR 16#1;
	ELSE
		T_Visu.ptrT_ExchgParam^.T_StationCommon.bStateMachine:=T_Visu.ptrT_ExchgParam^.T_StationCommon.bStateMachine AND 16#FE;
	END_IF;
	IF NOT(T_Station.TControl.xEnd) AND T_Station.TControl.xRdy AND T_Station.TControl.xEnable THEN
		T_Visu.ptrT_ExchgParam^.T_StationCommon.bStateMachine:=T_Visu.ptrT_ExchgParam^.T_StationCommon.bStateMachine OR 16#2;
	ELSE
		T_Visu.ptrT_ExchgParam^.T_StationCommon.bStateMachine:=T_Visu.ptrT_ExchgParam^.T_StationCommon.bStateMachine AND 16#FD;
	END_IF;
	IF T_Station.TControl.xError THEN
		T_Visu.ptrT_ExchgParam^.T_StationCommon.bStateMachine:=T_Visu.ptrT_ExchgParam^.T_StationCommon.bStateMachine OR 16#4;
	ELSE
		T_Visu.ptrT_ExchgParam^.T_StationCommon.bStateMachine:=T_Visu.ptrT_ExchgParam^.T_StationCommon.bStateMachine AND 16#FB;
	END_IF;
	IF T_Station.TControl.xReferenced THEN
		T_Visu.ptrT_ExchgParam^.T_StationCommon.bStateMachine:=T_Visu.ptrT_ExchgParam^.T_StationCommon.bStateMachine OR 16#8;
	ELSE
		T_Visu.ptrT_ExchgParam^.T_StationCommon.bStateMachine:=T_Visu.ptrT_ExchgParam^.T_StationCommon.bStateMachine AND 16#F7;
	END_IF;

(* Monitoring for the visu of the state of the machine *)
	T_Visu.ptrT_ExchgParam^.T_StationCommon.bStateMachineLED:=16#0;
	IF T_Station.TControl.xError OR T_Station.THardware.TAxisToolLeft.T_CtrleSingle.xErr OR (T_Station.THardware.TAxisToolCenter.T_CtrleSingle.xErr AND xMicroRodActive) OR
	    T_Station.THardware.TAxisToolRight.T_CtrleSingle.xErr OR T_Station.THardware.TAxisToolFeeder.T_CtrleSingle.xErr OR T_Station.THardware.TAxisGrindFeeder.T_CtrleSingle.xErr OR
	     (T_ExchgParam.T_Visu.T_Message.iState = 401) THEN
		T_Visu.ptrT_ExchgParam^.T_StationCommon.bStateMachineLED:=16#4;
	ELSIF NOT(T_Station.TControl.xEnd) OR NOT(T_Process.xEnd) OR T_Station.TControl.xActiveMovement THEN
		T_Visu.ptrT_ExchgParam^.T_StationCommon.bStateMachineLED:=16#2;
	ELSE
		T_Visu.ptrT_ExchgParam^.T_StationCommon.bStateMachineLED:=16#1;
	END_IF;
	IF (T_Visu.ptrT_ExchgParam^.T_StationCommon.bStateMachineLED <> 16#4) THEN
		IF NOT(T_TwinSafeOut.QxContactor_K3) OR NOT(T_TwinSafeOut.QxContactor_K4) THEN
			T_Visu.ptrT_ExchgParam^.T_StationCommon.bStateMachineLED:=16#0;
		END_IF;
	END_IF



(* Monitoring ActuatorState *)
Monitor_ActuatorState;



(* Bt Function panel *)
	(* Fn Bt function panel state *)
	CASE T_Visu.T_PlcParam.dwActualPage OF
	10:			wTmp:=16#0;
				IF T_Visu.ptrT_ExchgParam^.T_StationCommon.T_AutoGeometryPara.xPlungeActivationGeometry THEN wTmp:=wTmp+16#1; ELSE wTmp:=wTmp AND 16#FE; END_IF
				IF T_Visu.ptrT_ExchgParam^.T_StationCommon.T_AutoGeometryPara.xDisplaceActivationGeometry THEN wTmp:=wTmp+16#2; ELSE wTmp:=wTmp AND 16#FD; END_IF
				IF T_Visu.ptrT_ExchgParam^.T_Cylinder.xToolTension THEN wTmp:=wTmp+16#4; ELSE wTmp:=wTmp AND 16#FB; END_IF
				IF T_Visu.ptrT_ExchgParam^.T_StationCommon.T_AutoGeometryPara.xWarmUp THEN wTmp:=wTmp+16#20; ELSE wTmp:=wTmp AND 16#DF; END_IF
				xTmp:=	T_Station.THardware.TAxisToolLeft.T_CtrleSingle.xPower AND
						((T_Station.THardware.TAxisToolCenter.T_CtrleSingle.xPower AND xMicroRodActive) OR NOT(xMicroRodActive)) AND
						T_Station.THardware.TAxisToolRight.T_CtrleSingle.xPower AND
						T_Station.THardware.TAxisToolFeeder.T_CtrleSingle.xPower AND
						T_Station.THardware.TAxisGrindFeeder.T_CtrleSingle.xPower;
				IF xTmp THEN wTmp:=wTmp+16#8; ELSE wTmp:=wTmp AND 16#F7; END_IF
	20:			wTmp:=16#0;
				IF T_Visu.ptrT_ExchgParam^.T_StationCommon.T_AutoGroovePara.xPlungeActivationGroove THEN wTmp:=wTmp+16#1; ELSE wTmp:=wTmp AND 16#FE; END_IF
				IF T_Visu.ptrT_ExchgParam^.T_StationCommon.T_AutoGroovePara.xDisplaceActivationGroove THEN wTmp:=wTmp+16#2; ELSE wTmp:=wTmp AND 16#FD; END_IF
				IF T_Visu.ptrT_ExchgParam^.T_Cylinder.xToolTension THEN wTmp:=wTmp+16#4; ELSE wTmp:=wTmp AND 16#FB; END_IF
				IF T_Visu.ptrT_ExchgParam^.T_StationCommon.T_AutoGroovePara.xBlockGrindFeeder THEN wTmp:=wTmp+16#20; ELSE wTmp:=wTmp AND 16#DF; END_IF
	30:			wTmp:=16#0;
				IF T_Visu.ptrT_ExchgParam^.T_Cylinder.xToolTension THEN wTmp:=wTmp+16#4; ELSE wTmp:=wTmp AND 16#FB; END_IF
				xTmp:=	T_Station.THardware.TAxisToolLeft.T_CtrleSingle.xPower AND
						((T_Station.THardware.TAxisToolCenter.T_CtrleSingle.xPower AND xMicroRodActive) OR NOT(xMicroRodActive)) AND
						T_Station.THardware.TAxisToolRight.T_CtrleSingle.xPower AND
						T_Station.THardware.TAxisToolFeeder.T_CtrleSingle.xPower AND
						T_Station.THardware.TAxisGrindFeeder.T_CtrleSingle.xPower;
				IF xTmp THEN wTmp:=wTmp+16#8; ELSE wTmp:=wTmp AND 16#F7; END_IF
	110:			wTmp:=16#0;
				IF T_Visu.ptrT_ExchgParam^.T_StationCommon.T_CalibrationPara.xPlungeActivationCalib THEN wTmp:=wTmp+16#1; ELSE wTmp:=wTmp AND 16#FE; END_IF
				IF T_Visu.ptrT_ExchgParam^.T_StationCommon.T_CalibrationPara.xDisplaceActivationCalib THEN wTmp:=wTmp+16#2; ELSE wTmp:=wTmp AND 16#FD; END_IF
				IF T_Visu.ptrT_ExchgParam^.T_Cylinder.xToolTension THEN wTmp:=wTmp+16#4; ELSE wTmp:=wTmp AND 16#FB; END_IF
(*SOA 21.02.2023  {    *)
	141:			wTmp:=16#0;
				IF xStartUpConfirmed THEN wTmp:=wTmp+16#1; ELSE wTmp:=wTmp AND 16#FE; END_IF
(*SOA 21.02.2023  }   *)
	220:			wTmp:=16#0;
				IF T_Visu.ptrT_ExchgParam^.T_Cylinder.xToolTension THEN wTmp:=wTmp+16#4; ELSE wTmp:=wTmp AND 16#FB; END_IF
	310:			wTmp:=16#0;
				IF T_Visu.ptrT_ExchgParam^.T_Cylinder.xToolTension THEN wTmp:=wTmp+16#10; ELSE wTmp:=wTmp AND 16#EF; END_IF
	330:			wTmp:=16#0;
				IF T_Visu.ptrT_ExchgParam^.T_Cylinder.xToolTension THEN wTmp:=wTmp+16#10; ELSE wTmp:=wTmp AND 16#EF; END_IF
				xTmp:=	T_Station.THardware.TAxisToolLeft.T_CtrleSingle.xPower AND
						((T_Station.THardware.TAxisToolCenter.T_CtrleSingle.xPower AND xMicroRodActive) OR NOT(xMicroRodActive)) AND
						T_Station.THardware.TAxisToolRight.T_CtrleSingle.xPower AND
						T_Station.THardware.TAxisToolFeeder.T_CtrleSingle.xPower AND
						T_Station.THardware.TAxisGrindFeeder.T_CtrleSingle.xPower;
				IF xTmp THEN wTmp:=wTmp+16#1; ELSE wTmp:=wTmp AND 16#FE; END_IF
	410:			wTmp:=16#0;
				CASE T_Visu.ptrT_ExchgParam^.T_TeachIn.iSelectAxisGrind OF
				1:	;
				2:	IF QxGrindingSpindle_ReleaseBrake THEN	wTmp:=wTmp+16#20; ELSE wTmp:=wTmp AND 16#DF; END_IF
				END_CASE
	ELSE wTmp:=16#0;
	END_CASE
	T_Visu.ptrT_ExchgParam^.T_BtFunctionPanel.wState:=wTmp;

(* Monitoring ToolTorque *)
	IF (T_Visu.T_PlcParam.dwActualPage = 220) THEN
		T_Visu.ptrT_ExchgParam^.T_InfoValueCommon.rActualToolLeftTorque:=T_Station.THardware.TAxisToolLeft.T_LiveValue.uiActualTorque;
		T_Visu.ptrT_ExchgParam^.T_InfoValueCommon.rActualToolRightTorque:=T_Station.THardware.TAxisToolRight.T_LiveValue.uiActualTorque;
		T_Visu.ptrT_ExchgParam^.T_InfoValueCommon.rActualToolCenterTorque:=T_Station.THardware.TAxisToolCenter.T_LiveValue.uiActualTorque;
		FBCalcTorqueToolLeft(	xStart:=TRUE,
								uiActualTorque:= T_Station.THardware.TAxisToolLeft.T_LiveValue.uiActualTorque,
								uiZeroTorque:=uiToolLeftZeroTorque,
								iStepCalc:= 100);
		FBCalcTorqueToolCenter(	xStart:=TRUE,
								uiActualTorque:= T_Station.THardware.TAxisToolCenter.T_LiveValue.uiActualTorque,
								uiZeroTorque:=uiToolCenterZeroTorque,
								iStepCalc:= 100);
		FBCalcTorqueToolRight(	xStart:=TRUE,
								uiActualTorque:= T_Station.THardware.TAxisToolRight.T_LiveValue.uiActualTorque,
								uiZeroTorque:=uiToolRightZeroTorque,
								iStepCalc:= 100);
		T_Visu.ptrT_ExchgParam^.T_InfoValueCommon.rCalculToolLeftTorque:=FBCalcTorqueToolLeft.uiCalcTorque;
		T_Visu.ptrT_ExchgParam^.T_InfoValueCommon.rCalculToolCenterTorque:=FBCalcTorqueToolCenter.uiCalcTorque;
		T_Visu.ptrT_ExchgParam^.T_InfoValueCommon.rCalculToolRightTorque:=FBCalcTorqueToolRight.uiCalcTorque;
	ELSE
		FBCalcTorqueToolLeft(	xStart:=FALSE);
		FBCalcTorqueToolCenter(	xStart:=FALSE);
		FBCalcTorqueToolRight(	xStart:=FALSE);
	END_IF;

(* Monitoring Max ToolRotation Speed *)
	IF xMicroRodActive THEN
		T_Visu.ptrT_ExchgParam^.T_StationCommon.rMaxSpeedToolRotation:=1200.0;
	ELSE
		T_Visu.ptrT_ExchgParam^.T_StationCommon.rMaxSpeedToolRotation:=500.0;
	END_IF;

(* Monitoring AutoGeometry or AutoGroove *)
	IF (T_Visu.T_PlcParam.dwActualPage = 10) OR (T_Visu.T_PlcParam.dwActualPage = 20) THEN
		xPart1:=xPart2:=xPart3:=xPart4:=xPart5:=xPart6:=FALSE;
		rToolTotalLength:=0.0;
		IF T_Visu.ptrT_ExchgParam^.T_GeometryCommon.T_Geometry.axActiveSection[1] THEN
			xPart1:=TRUE;
			T_Visu.ptrT_ExchgParam^.T_InfoValueCommon.arStartDiameter[1]:=T_Visu.ptrT_ExchgParam^.T_GeometryCommon.T_Geometry.arStartDiameter[1];
			T_Visu.ptrT_ExchgParam^.T_InfoValueCommon.arEndDiameter[1]:=T_Visu.ptrT_ExchgParam^.T_GeometryCommon.T_Geometry.arEndDiameter[1];
			rToolTotalLength:=rToolTotalLength + T_Visu.ptrT_ExchgParam^.T_GeometryCommon.T_Geometry.arSectionLength[1];
			IF T_Visu.ptrT_ExchgParam^.T_GeometryCommon.T_Geometry.axActiveSection[2] THEN
				xPart2:=TRUE;
				T_Visu.ptrT_ExchgParam^.T_InfoValueCommon.arStartDiameter[2]:=T_Visu.ptrT_ExchgParam^.T_GeometryCommon.T_Geometry.arStartDiameter[2];
				T_Visu.ptrT_ExchgParam^.T_InfoValueCommon.arEndDiameter[2]:=T_Visu.ptrT_ExchgParam^.T_GeometryCommon.T_Geometry.arEndDiameter[2];
				rToolTotalLength:=rToolTotalLength + T_Visu.ptrT_ExchgParam^.T_GeometryCommon.T_Geometry.arSectionLength[2];
				IF T_Visu.ptrT_ExchgParam^.T_GeometryCommon.T_Geometry.axActiveSection[3] THEN
					xPart3:=TRUE;
					T_Visu.ptrT_ExchgParam^.T_InfoValueCommon.arStartDiameter[3]:=T_Visu.ptrT_ExchgParam^.T_GeometryCommon.T_Geometry.arStartDiameter[3];
					T_Visu.ptrT_ExchgParam^.T_InfoValueCommon.arEndDiameter[3]:=T_Visu.ptrT_ExchgParam^.T_GeometryCommon.T_Geometry.arEndDiameter[3];
					rToolTotalLength:=rToolTotalLength + T_Visu.ptrT_ExchgParam^.T_GeometryCommon.T_Geometry.arSectionLength[3];
					IF T_Visu.ptrT_ExchgParam^.T_GeometryCommon.T_Geometry.axActiveSection[4] THEN
						xPart4:=TRUE;
						T_Visu.ptrT_ExchgParam^.T_InfoValueCommon.arStartDiameter[4]:=T_Visu.ptrT_ExchgParam^.T_GeometryCommon.T_Geometry.arStartDiameter[4];
						T_Visu.ptrT_ExchgParam^.T_InfoValueCommon.arEndDiameter[4]:=T_Visu.ptrT_ExchgParam^.T_GeometryCommon.T_Geometry.arEndDiameter[4];
						rToolTotalLength:=rToolTotalLength + T_Visu.ptrT_ExchgParam^.T_GeometryCommon.T_Geometry.arSectionLength[4];
					(*09.12.2022: SOA	{	 *)
						IF T_Visu.ptrT_ExchgParam^.T_GeometryCommon.T_Geometry.axActiveSection[5] THEN
							xPart5:=TRUE;
							T_Visu.ptrT_ExchgParam^.T_InfoValueCommon.arStartDiameter[5]:=T_Visu.ptrT_ExchgParam^.T_GeometryCommon.T_Geometry.arStartDiameter[5];
							T_Visu.ptrT_ExchgParam^.T_InfoValueCommon.arEndDiameter[5]:=T_Visu.ptrT_ExchgParam^.T_GeometryCommon.T_Geometry.arEndDiameter[5];
							rToolTotalLength:=rToolTotalLength + T_Visu.ptrT_ExchgParam^.T_GeometryCommon.T_Geometry.arSectionLength[5];
							IF T_Visu.ptrT_ExchgParam^.T_GeometryCommon.T_Geometry.axActiveSection[6] THEN
								xPart6:=TRUE;
								T_Visu.ptrT_ExchgParam^.T_InfoValueCommon.arStartDiameter[6]:=T_Visu.ptrT_ExchgParam^.T_GeometryCommon.T_Geometry.arStartDiameter[6];
								T_Visu.ptrT_ExchgParam^.T_InfoValueCommon.arEndDiameter[6]:=T_Visu.ptrT_ExchgParam^.T_GeometryCommon.T_Geometry.arEndDiameter[6];
								rToolTotalLength:=rToolTotalLength + T_Visu.ptrT_ExchgParam^.T_GeometryCommon.T_Geometry.arSectionLength[6];
							END_IF;
						END_IF;
					(*09.12.2022: SOA	}	 *)
					END_IF;
				END_IF;
			END_IF;

		ELSIF T_Visu.ptrT_ExchgParam^.T_GeometryCommon.T_Geometry.axActiveSection[2] THEN
			xPart2:=TRUE;
			T_Visu.ptrT_ExchgParam^.T_InfoValueCommon.arStartDiameter[1]:=T_Visu.ptrT_ExchgParam^.T_GeometryCommon.T_Geometry.arStartDiameter[2];
			T_Visu.ptrT_ExchgParam^.T_InfoValueCommon.arEndDiameter[1]:=T_Visu.ptrT_ExchgParam^.T_GeometryCommon.T_Geometry.arEndDiameter[2];
			rToolTotalLength:=rToolTotalLength + T_Visu.ptrT_ExchgParam^.T_GeometryCommon.T_Geometry.arSectionLength[2];
			IF T_Visu.ptrT_ExchgParam^.T_GeometryCommon.T_Geometry.axActiveSection[3] THEN
				xPart3:=TRUE;
				T_Visu.ptrT_ExchgParam^.T_InfoValueCommon.arStartDiameter[2]:=T_Visu.ptrT_ExchgParam^.T_GeometryCommon.T_Geometry.arStartDiameter[3];
				T_Visu.ptrT_ExchgParam^.T_InfoValueCommon.arEndDiameter[2]:=T_Visu.ptrT_ExchgParam^.T_GeometryCommon.T_Geometry.arEndDiameter[3];
				rToolTotalLength:=rToolTotalLength + T_Visu.ptrT_ExchgParam^.T_GeometryCommon.T_Geometry.arSectionLength[3];
				IF T_Visu.ptrT_ExchgParam^.T_GeometryCommon.T_Geometry.axActiveSection[4] THEN
					xPart4:=TRUE;
					T_Visu.ptrT_ExchgParam^.T_InfoValueCommon.arStartDiameter[3]:=T_Visu.ptrT_ExchgParam^.T_GeometryCommon.T_Geometry.arStartDiameter[4];
					T_Visu.ptrT_ExchgParam^.T_InfoValueCommon.arEndDiameter[3]:=T_Visu.ptrT_ExchgParam^.T_GeometryCommon.T_Geometry.arEndDiameter[4];
					rToolTotalLength:=rToolTotalLength + T_Visu.ptrT_ExchgParam^.T_GeometryCommon.T_Geometry.arSectionLength[4];
					IF T_Visu.ptrT_ExchgParam^.T_GeometryCommon.T_Geometry.axActiveSection[5] THEN
						xPart5:=TRUE;
						T_Visu.ptrT_ExchgParam^.T_InfoValueCommon.arStartDiameter[4]:=T_Visu.ptrT_ExchgParam^.T_GeometryCommon.T_Geometry.arStartDiameter[5];
						T_Visu.ptrT_ExchgParam^.T_InfoValueCommon.arEndDiameter[4]:=T_Visu.ptrT_ExchgParam^.T_GeometryCommon.T_Geometry.arEndDiameter[5];
						rToolTotalLength:=rToolTotalLength + T_Visu.ptrT_ExchgParam^.T_GeometryCommon.T_Geometry.arSectionLength[5];
						IF T_Visu.ptrT_ExchgParam^.T_GeometryCommon.T_Geometry.axActiveSection[6] THEN
							xPart6:=TRUE;
							T_Visu.ptrT_ExchgParam^.T_InfoValueCommon.arStartDiameter[5]:=T_Visu.ptrT_ExchgParam^.T_GeometryCommon.T_Geometry.arStartDiameter[6];
							T_Visu.ptrT_ExchgParam^.T_InfoValueCommon.arEndDiameter[5]:=T_Visu.ptrT_ExchgParam^.T_GeometryCommon.T_Geometry.arEndDiameter[6];
							rToolTotalLength:=rToolTotalLength + T_Visu.ptrT_ExchgParam^.T_GeometryCommon.T_Geometry.arSectionLength[6];
						END_IF;
					END_IF;
				END_IF;
			END_IF;
		ELSIF T_Visu.ptrT_ExchgParam^.T_GeometryCommon.T_Geometry.axActiveSection[3] THEN
			xPart3:=TRUE;
			T_Visu.ptrT_ExchgParam^.T_InfoValueCommon.arStartDiameter[1]:=T_Visu.ptrT_ExchgParam^.T_GeometryCommon.T_Geometry.arStartDiameter[3];
			T_Visu.ptrT_ExchgParam^.T_InfoValueCommon.arEndDiameter[1]:=T_Visu.ptrT_ExchgParam^.T_GeometryCommon.T_Geometry.arEndDiameter[3];
			rToolTotalLength:=rToolTotalLength + T_Visu.ptrT_ExchgParam^.T_GeometryCommon.T_Geometry.arSectionLength[3];
			IF T_Visu.ptrT_ExchgParam^.T_GeometryCommon.T_Geometry.axActiveSection[4] THEN
				xPart4:=TRUE;
				T_Visu.ptrT_ExchgParam^.T_InfoValueCommon.arStartDiameter[2]:=T_Visu.ptrT_ExchgParam^.T_GeometryCommon.T_Geometry.arStartDiameter[4];
				T_Visu.ptrT_ExchgParam^.T_InfoValueCommon.arEndDiameter[2]:=T_Visu.ptrT_ExchgParam^.T_GeometryCommon.T_Geometry.arEndDiameter[4];
				rToolTotalLength:=rToolTotalLength + T_Visu.ptrT_ExchgParam^.T_GeometryCommon.T_Geometry.arSectionLength[4];
				IF T_Visu.ptrT_ExchgParam^.T_GeometryCommon.T_Geometry.axActiveSection[5] THEN
					xPart5:=TRUE;
					T_Visu.ptrT_ExchgParam^.T_InfoValueCommon.arStartDiameter[3]:=T_Visu.ptrT_ExchgParam^.T_GeometryCommon.T_Geometry.arStartDiameter[5];
					T_Visu.ptrT_ExchgParam^.T_InfoValueCommon.arEndDiameter[3]:=T_Visu.ptrT_ExchgParam^.T_GeometryCommon.T_Geometry.arEndDiameter[5];
					rToolTotalLength:=rToolTotalLength + T_Visu.ptrT_ExchgParam^.T_GeometryCommon.T_Geometry.arSectionLength[5];
					IF T_Visu.ptrT_ExchgParam^.T_GeometryCommon.T_Geometry.axActiveSection[6] THEN
						xPart6:=TRUE;
						T_Visu.ptrT_ExchgParam^.T_InfoValueCommon.arStartDiameter[4]:=T_Visu.ptrT_ExchgParam^.T_GeometryCommon.T_Geometry.arStartDiameter[6];
						T_Visu.ptrT_ExchgParam^.T_InfoValueCommon.arEndDiameter[4]:=T_Visu.ptrT_ExchgParam^.T_GeometryCommon.T_Geometry.arEndDiameter[6];
						rToolTotalLength:=rToolTotalLength + T_Visu.ptrT_ExchgParam^.T_GeometryCommon.T_Geometry.arSectionLength[6];
					END_IF;
				END_IF;
			END_IF;
		ELSIF T_Visu.ptrT_ExchgParam^.T_GeometryCommon.T_Geometry.axActiveSection[4] THEN
			xPart4:=TRUE;
			T_Visu.ptrT_ExchgParam^.T_InfoValueCommon.arStartDiameter[1]:=T_Visu.ptrT_ExchgParam^.T_GeometryCommon.T_Geometry.arStartDiameter[4];
			T_Visu.ptrT_ExchgParam^.T_InfoValueCommon.arEndDiameter[1]:=T_Visu.ptrT_ExchgParam^.T_GeometryCommon.T_Geometry.arEndDiameter[4];
			rToolTotalLength:=rToolTotalLength + T_Visu.ptrT_ExchgParam^.T_GeometryCommon.T_Geometry.arSectionLength[4];
			IF T_Visu.ptrT_ExchgParam^.T_GeometryCommon.T_Geometry.axActiveSection[5] THEN
				xPart5:=TRUE;
				T_Visu.ptrT_ExchgParam^.T_InfoValueCommon.arStartDiameter[2]:=T_Visu.ptrT_ExchgParam^.T_GeometryCommon.T_Geometry.arStartDiameter[5];
				T_Visu.ptrT_ExchgParam^.T_InfoValueCommon.arEndDiameter[2]:=T_Visu.ptrT_ExchgParam^.T_GeometryCommon.T_Geometry.arEndDiameter[5];
				rToolTotalLength:=rToolTotalLength + T_Visu.ptrT_ExchgParam^.T_GeometryCommon.T_Geometry.arSectionLength[5];
				IF T_Visu.ptrT_ExchgParam^.T_GeometryCommon.T_Geometry.axActiveSection[6] THEN
						xPart6:=TRUE;
						T_Visu.ptrT_ExchgParam^.T_InfoValueCommon.arStartDiameter[3]:=T_Visu.ptrT_ExchgParam^.T_GeometryCommon.T_Geometry.arStartDiameter[6];
						T_Visu.ptrT_ExchgParam^.T_InfoValueCommon.arEndDiameter[3]:=T_Visu.ptrT_ExchgParam^.T_GeometryCommon.T_Geometry.arEndDiameter[6];
						rToolTotalLength:=rToolTotalLength + T_Visu.ptrT_ExchgParam^.T_GeometryCommon.T_Geometry.arSectionLength[6];
				END_IF;
			END_IF;
		ELSIF T_Visu.ptrT_ExchgParam^.T_GeometryCommon.T_Geometry.axActiveSection[5] THEN
			xPart5:=TRUE;
			T_Visu.ptrT_ExchgParam^.T_InfoValueCommon.arStartDiameter[1]:=T_Visu.ptrT_ExchgParam^.T_GeometryCommon.T_Geometry.arStartDiameter[5];
			T_Visu.ptrT_ExchgParam^.T_InfoValueCommon.arEndDiameter[1]:=T_Visu.ptrT_ExchgParam^.T_GeometryCommon.T_Geometry.arEndDiameter[5];
			rToolTotalLength:=rToolTotalLength + T_Visu.ptrT_ExchgParam^.T_GeometryCommon.T_Geometry.arSectionLength[5];
			IF T_Visu.ptrT_ExchgParam^.T_GeometryCommon.T_Geometry.axActiveSection[6] THEN
				xPart6:=TRUE;
				T_Visu.ptrT_ExchgParam^.T_InfoValueCommon.arStartDiameter[2]:=T_Visu.ptrT_ExchgParam^.T_GeometryCommon.T_Geometry.arStartDiameter[6];
				T_Visu.ptrT_ExchgParam^.T_InfoValueCommon.arEndDiameter[2]:=T_Visu.ptrT_ExchgParam^.T_GeometryCommon.T_Geometry.arEndDiameter[6];
				rToolTotalLength:=rToolTotalLength + T_Visu.ptrT_ExchgParam^.T_GeometryCommon.T_Geometry.arSectionLength[6];
			END_IF;
		ELSIF T_Visu.ptrT_ExchgParam^.T_GeometryCommon.T_Geometry.axActiveSection[6] THEN
			xPart6:=TRUE;
			T_Visu.ptrT_ExchgParam^.T_InfoValueCommon.arStartDiameter[1]:=T_Visu.ptrT_ExchgParam^.T_GeometryCommon.T_Geometry.arStartDiameter[6];
			T_Visu.ptrT_ExchgParam^.T_InfoValueCommon.arEndDiameter[1]:=T_Visu.ptrT_ExchgParam^.T_GeometryCommon.T_Geometry.arEndDiameter[6];
			rToolTotalLength:=rToolTotalLength + T_Visu.ptrT_ExchgParam^.T_GeometryCommon.T_Geometry.arSectionLength[6];

		ELSE
			FOR ii:=1 TO 6 DO
				T_Visu.ptrT_ExchgParam^.T_InfoValueCommon.arStartDiameter[ii]:=0;
				T_Visu.ptrT_ExchgParam^.T_InfoValueCommon.arEndDiameter[ii]:=0;
			END_FOR;
		END_IF;
		iPartActive:=0;
		IF xPart1 THEN iPartActive:=iPartActive + 1; END_IF;
		IF xPart2 THEN iPartActive:=iPartActive + 1; END_IF;
		IF xPart3 THEN iPartActive:=iPartActive + 1; END_IF;
		IF xPart4 THEN iPartActive:=iPartActive + 1; END_IF;
		IF xPart5 THEN iPartActive:=iPartActive + 1; END_IF;
		IF xPart6 THEN iPartActive:=iPartActive + 1; END_IF;

		IF (iPartActive > 0) THEN
			FOR ii:=6 TO (iPartActive + 1) BY -1 DO
				T_Visu.ptrT_ExchgParam^.T_InfoValueCommon.arStartDiameter[ii]:=0;
				T_Visu.ptrT_ExchgParam^.T_InfoValueCommon.arEndDiameter[ii]:=0;
			END_FOR;
		END_IF;

		T_Visu.ptrT_ExchgParam^.T_InfoValueCommon.iTotalCountDownCycle:=T_NovRAM.T_Data.T_ProcessImageData.T_AutoGeometryPara.iCycleGeometry;
		T_Visu.ptrT_ExchgParam^.T_InfoValueCommon.iTotalCountDownPlungeCycle:=T_Station.T_WorkTool.iTotalCountDownPlungeCycle;
		T_Visu.ptrT_ExchgParam^.T_InfoValueCommon.iTotalCountDownGrooveCycle:=T_NovRAM.T_Data.T_ProcessImageData.T_AutoGroovePara.iNumberOfGrooves;
		T_Visu.ptrT_ExchgParam^.T_InfoValueCommon.rToolDiameter:=T_NovRAM.T_Data.T_ProcessImageData.T_ProcessPara.rToolDiameterProcess;
		T_Visu.ptrT_ExchgParam^.T_InfoValueCommon.rToolTotalLength:=rToolTotalLength * 10.0;	(* umwandeln von cm in mm *)
		IF (T_Visu.T_PlcParam.dwActualPage = 10) THEN
			IF T_NovRAM.T_Data.T_ProcessImageData.T_AutoGeometryPara.xPlungeActivationGeometry THEN
				T_Visu.ptrT_ExchgParam^.T_InfoValueCommon.rToolTotalLength:=T_Visu.ptrT_ExchgParam^.T_InfoValueCommon.rToolTotalLength + T_NovRAM.T_Data.T_ProcessImageData.T_AutoGeometryPara.rPlungeLengthToolFeedGeometry;
			END_IF;
			IF T_NovRAM.T_Data.T_ProcessImageData.T_AutoGeometryPara.xDisplaceActivationGeometry THEN
				T_Visu.ptrT_ExchgParam^.T_InfoValueCommon.rToolTotalLength:=T_Visu.ptrT_ExchgParam^.T_InfoValueCommon.rToolTotalLength + T_NovRAM.T_Data.T_ProcessImageData.T_AutoGeometryPara.rDisplaceLengthToolFeedGeometry;
			END_IF;
		END_IF;
		IF (T_Visu.T_PlcParam.dwActualPage = 20) THEN
			IF T_NovRAM.T_Data.T_ProcessImageData.T_AutoGroovePara.xPlungeActivationGroove AND NOT(T_NovRAM.T_Data.T_ProcessImageData.T_AutoGroovePara.xBlockGrindFeeder) THEN
				T_Visu.ptrT_ExchgParam^.T_InfoValueCommon.rToolTotalLength:=T_Visu.ptrT_ExchgParam^.T_InfoValueCommon.rToolTotalLength + T_NovRAM.T_Data.T_ProcessImageData.T_AutoGroovePara.rPlungeLengthToolFeedGroove;
			END_IF;
			IF T_NovRAM.T_Data.T_ProcessImageData.T_AutoGroovePara.xDisplaceActivationGroove THEN
				T_Visu.ptrT_ExchgParam^.T_InfoValueCommon.rToolTotalLength:=T_Visu.ptrT_ExchgParam^.T_InfoValueCommon.rToolTotalLength + T_NovRAM.T_Data.T_ProcessImageData.T_AutoGroovePara.rDisplaceLengthToolFeedGroove;
			END_IF;
		END_IF;
	ELSE
		T_Visu.ptrT_ExchgParam^.T_InfoValueCommon.iCountDownCycle:=1;
		T_Visu.ptrT_ExchgParam^.T_InfoValueCommon.iCountDownPlungeCycle:=1;
		T_Visu.ptrT_ExchgParam^.T_InfoValueCommon.iCountDownGrooveCycle:=1;
	END_IF;

(* Tool Geometry Managment *)
	IF (T_Visu.T_PlcParam.dwActualPage = 120) OR (T_Visu.T_PlcParam.dwActualPage = 121) THEN
		FailingEdgeGeometryManagement(CLK:=TRUE);
		RisingEdgeGeometryManagement(CLK:=(T_Visu.T_PlcParam.dwActualPage = 120) OR (T_Visu.T_PlcParam.dwActualPage = 121));
		IF RisingEdgeGeometryManagement.Q THEN
			arSaveToolGeometry:=T_Visu.ptrT_ExchgParam^.T_GeometryCommon.T_Geometry;
		END_IF;
		T_Visu.ptrT_ExchgParam^.T_GeometryCommon.rMinToolDiameter:=T_Visu.ptrT_ExchgParam^.T_StationCommon.T_PrismPara.rToolDiameterMin;
		T_Visu.ptrT_ExchgParam^.T_GeometryCommon.rMaxToolDiameter:=T_Visu.ptrT_ExchgParam^.T_StationCommon.T_PrismPara.rToolDiameterMax;
		T_Visu.ptrT_ExchgParam^.T_GeometryCommon.rMinToolLength:=0.1;
		T_Visu.ptrT_ExchgParam^.T_GeometryCommon.rMaxToolLength:=T_Visu.ptrT_ExchgParam^.T_StationCommon.rConfigMaxToolLength;

		IF (arSaveToolGeometry.arEndDiameter[1] <> T_Visu.ptrT_ExchgParam^.T_GeometryCommon.T_Geometry.arEndDiameter[1]) THEN
			arSaveToolGeometry.arEndDiameter[1]:=T_Visu.ptrT_ExchgParam^.T_GeometryCommon.T_Geometry.arEndDiameter[1];
			arSaveToolGeometry.arStartDiameter[2]:=arSaveToolGeometry.arEndDiameter[1];
			T_Visu.ptrT_ExchgParam^.T_GeometryCommon.T_Geometry.arStartDiameter[2]:=arSaveToolGeometry.arStartDiameter[2];
		END_IF;
		IF (arSaveToolGeometry.arStartDiameter[2] <> T_Visu.ptrT_ExchgParam^.T_GeometryCommon.T_Geometry.arStartDiameter[2]) THEN
			arSaveToolGeometry.arStartDiameter[2]:=T_Visu.ptrT_ExchgParam^.T_GeometryCommon.T_Geometry.arStartDiameter[2];
			arSaveToolGeometry.arEndDiameter[1]:=arSaveToolGeometry.arStartDiameter[2];
			T_Visu.ptrT_ExchgParam^.T_GeometryCommon.T_Geometry.arEndDiameter[1]:=arSaveToolGeometry.arEndDiameter[1];
		END_IF;
		IF (arSaveToolGeometry.arEndDiameter[2] <> T_Visu.ptrT_ExchgParam^.T_GeometryCommon.T_Geometry.arEndDiameter[2]) THEN
			arSaveToolGeometry.arEndDiameter[2]:=T_Visu.ptrT_ExchgParam^.T_GeometryCommon.T_Geometry.arEndDiameter[2];
			arSaveToolGeometry.arStartDiameter[3]:=arSaveToolGeometry.arEndDiameter[2];
			T_Visu.ptrT_ExchgParam^.T_GeometryCommon.T_Geometry.arStartDiameter[3]:=arSaveToolGeometry.arStartDiameter[3];
		END_IF;
		IF (arSaveToolGeometry.arStartDiameter[3] <> T_Visu.ptrT_ExchgParam^.T_GeometryCommon.T_Geometry.arStartDiameter[3]) THEN
			arSaveToolGeometry.arStartDiameter[3]:=T_Visu.ptrT_ExchgParam^.T_GeometryCommon.T_Geometry.arStartDiameter[3];
			arSaveToolGeometry.arEndDiameter[2]:=arSaveToolGeometry.arStartDiameter[3];
			T_Visu.ptrT_ExchgParam^.T_GeometryCommon.T_Geometry.arEndDiameter[2]:=arSaveToolGeometry.arEndDiameter[2];
		END_IF;
		IF (arSaveToolGeometry.arEndDiameter[3] <> T_Visu.ptrT_ExchgParam^.T_GeometryCommon.T_Geometry.arEndDiameter[3]) THEN
			arSaveToolGeometry.arEndDiameter[3]:=T_Visu.ptrT_ExchgParam^.T_GeometryCommon.T_Geometry.arEndDiameter[3];
			arSaveToolGeometry.arStartDiameter[4]:=arSaveToolGeometry.arEndDiameter[3];
			T_Visu.ptrT_ExchgParam^.T_GeometryCommon.T_Geometry.arStartDiameter[4]:=arSaveToolGeometry.arStartDiameter[4];
		END_IF;
		IF (arSaveToolGeometry.arStartDiameter[4] <> T_Visu.ptrT_ExchgParam^.T_GeometryCommon.T_Geometry.arStartDiameter[4]) THEN
			arSaveToolGeometry.arStartDiameter[4]:=T_Visu.ptrT_ExchgParam^.T_GeometryCommon.T_Geometry.arStartDiameter[4];
			arSaveToolGeometry.arEndDiameter[3]:=arSaveToolGeometry.arStartDiameter[4];
			T_Visu.ptrT_ExchgParam^.T_GeometryCommon.T_Geometry.arEndDiameter[3]:=arSaveToolGeometry.arEndDiameter[3];
		END_IF;
(*09.12.2022: SOA	{	 *)
		IF (arSaveToolGeometry.arEndDiameter[4] <> T_Visu.ptrT_ExchgParam^.T_GeometryCommon.T_Geometry.arEndDiameter[4]) THEN
			arSaveToolGeometry.arEndDiameter[4]:=T_Visu.ptrT_ExchgParam^.T_GeometryCommon.T_Geometry.arEndDiameter[4];
			arSaveToolGeometry.arStartDiameter[5]:=arSaveToolGeometry.arEndDiameter[4];
			T_Visu.ptrT_ExchgParam^.T_GeometryCommon.T_Geometry.arStartDiameter[5]:=arSaveToolGeometry.arStartDiameter[5];
		END_IF;
		IF (arSaveToolGeometry.arStartDiameter[5] <> T_Visu.ptrT_ExchgParam^.T_GeometryCommon.T_Geometry.arStartDiameter[5]) THEN
			arSaveToolGeometry.arStartDiameter[5]:=T_Visu.ptrT_ExchgParam^.T_GeometryCommon.T_Geometry.arStartDiameter[5];
			arSaveToolGeometry.arEndDiameter[4]:=arSaveToolGeometry.arStartDiameter[5];
			T_Visu.ptrT_ExchgParam^.T_GeometryCommon.T_Geometry.arEndDiameter[4]:=arSaveToolGeometry.arEndDiameter[4];
		END_IF;
		IF (arSaveToolGeometry.arEndDiameter[5] <> T_Visu.ptrT_ExchgParam^.T_GeometryCommon.T_Geometry.arEndDiameter[5]) THEN
			arSaveToolGeometry.arEndDiameter[5]:=T_Visu.ptrT_ExchgParam^.T_GeometryCommon.T_Geometry.arEndDiameter[5];
			arSaveToolGeometry.arStartDiameter[6]:=arSaveToolGeometry.arEndDiameter[5];
			T_Visu.ptrT_ExchgParam^.T_GeometryCommon.T_Geometry.arStartDiameter[6]:=arSaveToolGeometry.arStartDiameter[6];
		END_IF;
		IF (arSaveToolGeometry.arStartDiameter[6] <> T_Visu.ptrT_ExchgParam^.T_GeometryCommon.T_Geometry.arStartDiameter[6]) THEN
			arSaveToolGeometry.arStartDiameter[6]:=T_Visu.ptrT_ExchgParam^.T_GeometryCommon.T_Geometry.arStartDiameter[6];
			arSaveToolGeometry.arEndDiameter[5]:=arSaveToolGeometry.arStartDiameter[6];
			T_Visu.ptrT_ExchgParam^.T_GeometryCommon.T_Geometry.arEndDiameter[5]:=arSaveToolGeometry.arEndDiameter[5];
		END_IF;
(*09.12.2022: SOA	}	 *)

(*Select Form*)
		FOR ii:=1 TO 6 DO
			IF NOT(T_Visu.ptrT_ExchgParam^.T_GeometryCommon.T_Geometry.axActiveSection[ii]) THEN
				T_Visu.ptrT_ExchgParam^.T_GeometryCommon.abSectionSelectForm[ii]:=0;
			END_IF;
		END_FOR;
		FOR ii:=1 TO 6 DO
			IF (T_Visu.ptrT_ExchgParam^.T_GeometryCommon.T_Geometry.arStartDiameter[ii] = T_Visu.ptrT_ExchgParam^.T_GeometryCommon.T_Geometry.arEndDiameter[ii]) THEN
				IF T_Visu.ptrT_ExchgParam^.T_GeometryCommon.T_Geometry.axActiveSection[ii] THEN
					T_Visu.ptrT_ExchgParam^.T_GeometryCommon.abSectionSelectForm[ii]:=2;
				END_IF;
			END_IF;
		END_FOR;
		FOR ii:=1 TO 6 DO
			IF (T_Visu.ptrT_ExchgParam^.T_GeometryCommon.T_Geometry.arStartDiameter[ii] > T_Visu.ptrT_ExchgParam^.T_GeometryCommon.T_Geometry.arEndDiameter[ii]) THEN
				IF T_Visu.ptrT_ExchgParam^.T_GeometryCommon.T_Geometry.axActiveSection[ii] THEN
					T_Visu.ptrT_ExchgParam^.T_GeometryCommon.abSectionSelectForm[ii]:=3;
				END_IF;
			END_IF;
		END_FOR;
		FOR ii:=1 TO 6 DO
			IF (T_Visu.ptrT_ExchgParam^.T_GeometryCommon.T_Geometry.arStartDiameter[ii] < T_Visu.ptrT_ExchgParam^.T_GeometryCommon.T_Geometry.arEndDiameter[ii]) THEN
				IF T_Visu.ptrT_ExchgParam^.T_GeometryCommon.T_Geometry.axActiveSection[ii] THEN
					T_Visu.ptrT_ExchgParam^.T_GeometryCommon.abSectionSelectForm[ii]:=4;
				END_IF;
			END_IF;
		END_FOR;

 (*Checking for forbidden ToolDiameter - if forbidden: Set Bit in Word *)
	rCalcTotalToolLength:=0.0;
		FOR ii:=1 TO 6 DO
			IF ii>=1 AND ii<=4 THEN
				IF (T_Visu.ptrT_ExchgParam^.T_GeometryCommon.T_Geometry.arStartDiameter[ii] = 0) OR
				     (T_Visu.ptrT_ExchgParam^.T_GeometryCommon.T_Geometry.arStartDiameter[ii] > T_Visu.ptrT_ExchgParam^.T_StationCommon.T_PrismPara.rToolDiameterMax) OR
				     (T_Visu.ptrT_ExchgParam^.T_GeometryCommon.T_Geometry.arStartDiameter[ii] < T_Visu.ptrT_ExchgParam^.T_StationCommon.T_PrismPara.rToolDiameterMin) THEN
					T_Visu.ptrT_ExchgParam^.T_GeometryCommon.wWrongInput:=DWORD_TO_WORD(SETBIT32(T_Visu.ptrT_ExchgParam^.T_GeometryCommon.wWrongInput,INT_TO_SINT(ii-1)));
				ELSE
					T_Visu.ptrT_ExchgParam^.T_GeometryCommon.wWrongInput:=DWORD_TO_WORD(CLEARBIT32(T_Visu.ptrT_ExchgParam^.T_GeometryCommon.wWrongInput,INT_TO_SINT(ii-1)));
				END_IF;
				IF (T_Visu.ptrT_ExchgParam^.T_GeometryCommon.T_Geometry.arEndDiameter[ii] = 0) OR
				     (T_Visu.ptrT_ExchgParam^.T_GeometryCommon.T_Geometry.arEndDiameter[ii] > T_Visu.ptrT_ExchgParam^.T_StationCommon.T_PrismPara.rToolDiameterMax) OR
				     (T_Visu.ptrT_ExchgParam^.T_GeometryCommon.T_Geometry.arEndDiameter[ii] < T_Visu.ptrT_ExchgParam^.T_StationCommon.T_PrismPara.rToolDiameterMin) THEN
					T_Visu.ptrT_ExchgParam^.T_GeometryCommon.wWrongInput:=DWORD_TO_WORD(SETBIT32(T_Visu.ptrT_ExchgParam^.T_GeometryCommon.wWrongInput,INT_TO_SINT(ii+3)));
				ELSE
					T_Visu.ptrT_ExchgParam^.T_GeometryCommon.wWrongInput:=DWORD_TO_WORD(CLEARBIT32(T_Visu.ptrT_ExchgParam^.T_GeometryCommon.wWrongInput,INT_TO_SINT(ii+3)));
				END_IF;
				IF (T_Visu.ptrT_ExchgParam^.T_GeometryCommon.T_Geometry.arSectionPitch[ii] = 0) THEN
					T_Visu.ptrT_ExchgParam^.T_GeometryCommon.wWrongInput:=DWORD_TO_WORD(SETBIT32(T_Visu.ptrT_ExchgParam^.T_GeometryCommon.wWrongInput,INT_TO_SINT(ii+7)));
				ELSE
					T_Visu.ptrT_ExchgParam^.T_GeometryCommon.wWrongInput:=DWORD_TO_WORD(CLEARBIT32(T_Visu.ptrT_ExchgParam^.T_GeometryCommon.wWrongInput,INT_TO_SINT(ii+7)));
				END_IF;
				IF (T_Visu.ptrT_ExchgParam^.T_GeometryCommon.T_Geometry.arSectionLength[ii] = 0) THEN
					T_Visu.ptrT_ExchgParam^.T_GeometryCommon.wWrongInput:=DWORD_TO_WORD(SETBIT32(T_Visu.ptrT_ExchgParam^.T_GeometryCommon.wWrongInput,INT_TO_SINT(ii+11)));
				ELSE
					T_Visu.ptrT_ExchgParam^.T_GeometryCommon.wWrongInput:=DWORD_TO_WORD(CLEARBIT32(T_Visu.ptrT_ExchgParam^.T_GeometryCommon.wWrongInput,INT_TO_SINT(ii+11)));
				END_IF;
 (*09.12.2022: SOA *) (*Definition of second variable = wWrongInput_2*)
			ELSIF  ii>=5 AND ii<=6 THEN
				IF (T_Visu.ptrT_ExchgParam^.T_GeometryCommon.T_Geometry.arSectionPitch[ii] = 0) THEN
					T_Visu.ptrT_ExchgParam^.T_GeometryCommon.wWrongInput_2:=DWORD_TO_WORD(SETBIT32(T_Visu.ptrT_ExchgParam^.T_GeometryCommon.wWrongInput_2,INT_TO_SINT(ii-5)));
				ELSE
					T_Visu.ptrT_ExchgParam^.T_GeometryCommon.wWrongInput_2:=DWORD_TO_WORD(CLEARBIT32(T_Visu.ptrT_ExchgParam^.T_GeometryCommon.wWrongInput_2,INT_TO_SINT(ii-5)));
				END_IF;
				IF (T_Visu.ptrT_ExchgParam^.T_GeometryCommon.T_Geometry.arSectionLength[ii] = 0) THEN
					T_Visu.ptrT_ExchgParam^.T_GeometryCommon.wWrongInput_2:=DWORD_TO_WORD(SETBIT32(T_Visu.ptrT_ExchgParam^.T_GeometryCommon.wWrongInput_2,INT_TO_SINT(ii-1)));
				ELSE
					T_Visu.ptrT_ExchgParam^.T_GeometryCommon.wWrongInput_2:=DWORD_TO_WORD(CLEARBIT32(T_Visu.ptrT_ExchgParam^.T_GeometryCommon.wWrongInput_2,INT_TO_SINT(ii-1)));
				END_IF;
			END_IF;

			IF T_Visu.ptrT_ExchgParam^.T_GeometryCommon.T_Geometry.axActiveSection[ii] THEN
				rCalcTotalToolLength:=rCalcTotalToolLength + T_Visu.ptrT_ExchgParam^.T_GeometryCommon.T_Geometry.arSectionLength[ii];
			END_IF;
		END_FOR;

 (*Checking  every Section for active Bits, changing "SelectForm" if active *)
		IF (rCalcTotalToolLength > T_Visu.ptrT_ExchgParam^.T_StationCommon.rConfigMaxToolLength) AND ((T_Visu.ptrT_ExchgParam^.T_GeometryCommon.wWrongInput AND 16#F000) = 0) THEN
			T_Visu.ptrT_ExchgParam^.T_GeometryCommon.wWrongInput:=T_Visu.ptrT_ExchgParam^.T_GeometryCommon.wWrongInput OR 16#F000;
		END_IF;
		IF T_Visu.ptrT_ExchgParam^.T_GeometryCommon.T_Geometry.axActiveSection[1] THEN
			IF ((T_Visu.ptrT_ExchgParam^.T_GeometryCommon.wWrongInput AND 16#1111) <> 0) THEN
				T_Visu.ptrT_ExchgParam^.T_GeometryCommon.abSectionSelectForm[1]:=5;
			END_IF;
		END_IF;
		IF T_Visu.ptrT_ExchgParam^.T_GeometryCommon.T_Geometry.axActiveSection[2] THEN
			IF ((T_Visu.ptrT_ExchgParam^.T_GeometryCommon.wWrongInput AND 16#2222) <> 0) THEN
				T_Visu.ptrT_ExchgParam^.T_GeometryCommon.abSectionSelectForm[2]:=5;
			END_IF;
		END_IF;
		IF T_Visu.ptrT_ExchgParam^.T_GeometryCommon.T_Geometry.axActiveSection[3] THEN
			IF ((T_Visu.ptrT_ExchgParam^.T_GeometryCommon.wWrongInput AND 16#4444) <> 0) THEN
				T_Visu.ptrT_ExchgParam^.T_GeometryCommon.abSectionSelectForm[3]:=5;
			END_IF;
		END_IF;
		IF T_Visu.ptrT_ExchgParam^.T_GeometryCommon.T_Geometry.axActiveSection[4] THEN
			IF ((T_Visu.ptrT_ExchgParam^.T_GeometryCommon.wWrongInput AND 16#8888) <> 0) THEN
				T_Visu.ptrT_ExchgParam^.T_GeometryCommon.abSectionSelectForm[4]:=5;
			END_IF;
		END_IF;
(*09.12.2022: SOA	}	 *)
		IF T_Visu.ptrT_ExchgParam^.T_GeometryCommon.T_Geometry.axActiveSection[5] THEN
			IF ((T_Visu.ptrT_ExchgParam^.T_GeometryCommon.wWrongInput_2 AND 16#1111) <> 0) THEN
				T_Visu.ptrT_ExchgParam^.T_GeometryCommon.abSectionSelectForm[5]:=5;
			END_IF;
		END_IF;
		IF T_Visu.ptrT_ExchgParam^.T_GeometryCommon.T_Geometry.axActiveSection[6] THEN
			IF ((T_Visu.ptrT_ExchgParam^.T_GeometryCommon.wWrongInput_2 AND 16#2222) <> 0) THEN
				T_Visu.ptrT_ExchgParam^.T_GeometryCommon.abSectionSelectForm[6]:=5;
			END_IF;
		END_IF;
(*09.12.2022: SOA	}	 *)

	ELSE
		RisingEdgeGeometryManagement(CLK:=FALSE);
		FailingEdgeGeometryManagement(CLK:=FALSE);
		(*If the page changes, then copy again the settled value *)
		IF FailingEdgeGeometryManagement.Q THEN
			T_Visu.ptrT_ExchgParam^.T_GeometryCommon.T_Geometry:=T_NovRAM.T_Data.T_ProcessImageData.T_GeometryPara;
		END_IF;
	END_IF;

(* Monitoring Tool Geometry and Tool Calibration calculation Parameter *)
	T_Station.T_WorkTool.iBaseGearDivider:=15000;
	T_Station.T_WorkTool.rPrismaFactor:=T_NovRAM.T_Data.T_ProcessImageData.T_PrismPara.rPrismaFactor;
	T_Station.T_WorkTool.rGrindFeederScaleFactor:=T_Station.THardware.TAxisGrindFeeder.T_CtrleSingle.lrScaleFactor;
	T_Station.T_WorkTool.rToolFeederGearRatio:=T_Station.THardware.TAxisToolFeeder.T_CtrleSingle.lrGearRatio;
	T_Station.T_WorkTool.rToolFeederScaleFactor:=T_Station.THardware.TAxisToolFeeder.T_CtrleSingle.lrScaleFactor;
	T_Station.T_WorkTool.rToolRightGearRatio:=T_Station.THardware.TAxisToolRight.T_CtrleSingle.lrGearRatio;
	IF (T_Visu.T_PlcParam.dwActualPage = 10) OR (T_Visu.T_PlcParam.dwActualPage = 20) THEN
		IF (T_Visu.T_PlcParam.dwActualPage = 10) THEN
			iAutoProcess:=1;
			rToolRotationSpeed:=T_NovRAM.T_Data.T_ProcessImageData.T_AutoGeometryPara.rSpeedToolRotationGeometry;
			T_Station.T_WorkTool.rPlungeSpeedGrindFeed:=T_NovRAM.T_Data.T_ProcessImageData.T_AutoGeometryPara.rPlungeSpeedGrindFeedGeometry;
			T_Station.T_WorkTool.rDisplaceSpeedGrindFeed:=T_NovRAM.T_Data.T_ProcessImageData.T_AutoGeometryPara.rDisplaceSpeedGrindFeedGeometry;
		END_IF;
		IF (T_Visu.T_PlcParam.dwActualPage = 20) THEN
			iAutoProcess:=2;
			rToolRotationSpeed:=T_NovRAM.T_Data.T_ProcessImageData.T_AutoGroovePara.rSpeedToolRotationGroove;
			T_Station.T_WorkTool.rPlungeSpeedGrindFeed:=T_NovRAM.T_Data.T_ProcessImageData.T_AutoGroovePara.rPlungeSpeedGrindFeedGroove;
			T_Station.T_WorkTool.rDisplaceSpeedGrindFeed:=T_NovRAM.T_Data.T_ProcessImageData.T_AutoGroovePara.rDisplaceSpeedGrindFeedGroove;
		END_IF;
	ELSE
		iAutoProcess:=0;
	END_IF;
	IF (((T_Visu.T_PlcParam.dwActualPage = 10) OR (T_Visu.T_PlcParam.dwActualPage = 20) OR (T_Visu.T_PlcParam.dwActualPage = 110)) OR xCalcAgainProcTime) AND T_Visu.T_CtrleVisu.xDone THEN
		IF NOT(xCalcFirstTime) OR xCalcAgainProcTime THEN
			xCalcFirstTime:=TRUE;
			FBCalcProcessTime(	T_Geometry:=T_NovRAM.T_Data.T_ProcessImageData.T_GeometryPara,
								T_AutoGeometryPara:=T_NovRAM.T_Data.T_ProcessImageData.T_AutoGeometryPara,
								T_CalibrationPara:=T_NovRAM.T_Data.T_ProcessImageData.T_CalibrationPara,
								T_AutoGroovePara:=T_NovRAM.T_Data.T_ProcessImageData.T_AutoGroovePara,
								T_ProcessPara:=T_NovRAM.T_Data.T_ProcessImageData.T_ProcessPara,
								rToolRotationSpeed:=rToolRotationSpeed,
								rToolDiameter:=T_NovRAM.T_Data.T_ProcessImageData.T_ProcessPara.rToolDiameterProcess,
								rToolDiameterWithOffset:=	T_NovRAM.T_Data.T_ProcessImageData.T_ProcessPara.rToolDiameterProcess +
														T_NovRAM.T_Data.T_ProcessImageData.T_ProcessPara.rOffsetBeforeToolDiaGrindFeedProcess,
								iAutoProcess:=iAutoProcess,
								xMicroRodActive:=xMicroRodActive,
								T_WorkTool:=T_Station.T_WorkTool);
		END_IF;
		xCalcAgainProcTime:=FALSE;
		rAutoTimeTotal:=FBCalcProcessTime.rProcessTime;
		T_Visu.ptrT_ExchgParam^.T_InfoValueCommon.tAutoTimeTotal:=REAL_TO_TIME(rAutoTimeTotal * 1000.0);
	ELSE
		xCalcFirstTime:=FALSE;
	END_IF;
	IF T_Process.xEnd OR T_Process.xError THEN
		T_Visu.ptrT_ExchgParam^.T_InfoValueCommon.tAutoTimeLeft:=T_Visu.ptrT_ExchgParam^.T_InfoValueCommon.tAutoTimeTotal;
		T_Visu.ptrT_ExchgParam^.T_InfoValueCommon.bProgressbarAutoGeometry:=0;
		T_Visu.ptrT_ExchgParam^.T_InfoValueCommon.bProgressbarAutoGroove:=0;
		T_Visu.ptrT_ExchgParam^.T_InfoValueCommon.bProgressbarToolCalibration:=0;
	END_IF;

(* Monitoring ToolCalibration *)
	IF (T_Visu.T_PlcParam.dwActualPage = 110) THEN
		T_Visu.ptrT_ExchgParam^.T_InfoValueCommon.rToolLengthCalibration:=T_NovRAM.T_Data.T_ProcessImageData.T_CalibrationPara.rToolLengthCylinderPartCalib;
		T_Visu.ptrT_ExchgParam^.T_InfoValueCommon.rToolDiameter:=T_NovRAM.T_Data.T_ProcessImageData.T_ProcessPara.rToolDiameterProcess;
		T_Visu.ptrT_ExchgParam^.T_InfoValueCommon.rPitchCalibration:=T_NovRAM.T_Data.T_ProcessImageData.T_CalibrationPara.rPitchCalib;
	END_IF;

(* Monitoring Correction Tool Diameter *)
	IF (T_Visu.T_PlcParam.dwActualPage = 420) OR (T_Visu.T_PlcParam.dwActualPage = 11) OR (T_Visu.T_PlcParam.dwActualPage = 21) THEN
		RisingEdgeToolDiameter(CLK:=(T_Visu.T_PlcParam.dwActualPage = 420) OR (T_Visu.T_PlcParam.dwActualPage = 11) OR (T_Visu.T_PlcParam.dwActualPage = 21));
		IF RisingEdgeToolDiameter.Q THEN
			T_Visu.ptrT_ExchgParam^.T_InfoValueCommon.rCorrectionToolDiameter:=0.0;
			T_Visu.ptrT_ExchgParam^.T_InfoValueCommon.xKeyPadActivation:=FALSE;
		END_IF;
		IF (T_Visu.ptrT_ExchgParam^.T_InfoValueCommon.rCorrectionToolDiameter = 0) THEN
			T_Visu.ptrT_ExchgParam^.T_StationCommon.bStateToolDiameter:=1;
		END_IF;
		IF (T_Visu.ptrT_ExchgParam^.T_InfoValueCommon.rCorrectionToolDiameter > 0) THEN
			T_Visu.ptrT_ExchgParam^.T_StationCommon.bStateToolDiameter:=3;
		END_IF;
		IF (T_Visu.ptrT_ExchgParam^.T_InfoValueCommon.rCorrectionToolDiameter < 0) THEN
			T_Visu.ptrT_ExchgParam^.T_StationCommon.bStateToolDiameter:=2;
		END_IF;
	ELSE
		RisingEdgeToolDiameter(CLK:=FALSE);
	END_IF

(* Monitoring TeachIn Tool Rotation *)
	IF (T_Visu.T_PlcParam.dwActualPage = 210) THEN
		IF xToolRotationMasterSlave THEN
			T_Visu.ptrT_ExchgParam^.T_TeachIn.iSelectAxisToolRotation:=1;	(* Force Selection by choice of MasterSlave to the ToolLeft TouchButton *)
		END_IF;
		IF (T_Visu.ptrT_ExchgParam^.T_SafetyCtrl.bStateTeachInToolLeft = 2) OR (T_Visu.ptrT_ExchgParam^.T_SafetyCtrl.bStateTeachInToolCenter = 2) OR
		     (T_Visu.ptrT_ExchgParam^.T_SafetyCtrl.bStateTeachInToolRight = 2) THEN
			T_Visu.ptrT_ExchgParam^.T_TeachIn.iSelectAxisToolRotation:=iSelectAxisToolRotation;	(* Force Selection by active movement *)
		END_IF;
		IF (T_Visu.ptrT_ExchgParam^.T_TeachIn.iSelectAxisToolRotation <> iSelectAxisToolRotation) THEN
			iSelectAxisToolRotation:=T_Visu.ptrT_ExchgParam^.T_TeachIn.iSelectAxisToolRotation;
		END_IF;
	END_IF;
	IF (T_Visu.T_PlcParam.dwActualPage <> 210) AND xToolRotationMasterSlave THEN
		xToolRotationMasterSlave:=FALSE;
		IF xMicroRodActive THEN
			IF T_Station.THardware.TAxisToolCenter.T_CtrleSingle.xSlave AND T_Station.THardware.TAxisToolCenter.T_CtrleSingle.xDone THEN
				T_Station.THardware.TAxisToolCenter.T_CtrleSingle.iFunction:=25;
				T_Station.THardware.TAxisToolCenter.T_CtrleSingle.xExecute:=TRUE;
			END_IF;
		END_IF;
		IF T_Station.THardware.TAxisToolRight.T_CtrleSingle.xSlave AND T_Station.THardware.TAxisToolRight.T_CtrleSingle.xDone THEN
			T_Station.THardware.TAxisToolRight.T_CtrleSingle.iFunction:=25;
			T_Station.THardware.TAxisToolRight.T_CtrleSingle.xExecute:=TRUE;
		END_IF;
		IF NOT(xMicroRodActive) THEN
			IF T_Station.THardware.TAxisToolFeeder.T_CtrleSingle.xSlave AND T_Station.THardware.TAxisToolFeeder.T_CtrleSingle.xDone THEN
				T_Station.THardware.TAxisToolFeeder.T_CtrleSingle.iFunction:=25;
				T_Station.THardware.TAxisToolFeeder.T_CtrleSingle.xExecute:=TRUE;
			END_IF;
		END_IF;
	END_IF;

